LIN {X 0,Y 240.142,Z 967.676,A -85,B 0,C 180,E1 11583.81,E2 11583.81} C_VEL
LIN {X 0,Y 246.627,Z 959.065,A -85,B 0,C 180,E1 11579.011,E2 11579.011} C_VEL
LIN {X 0,Y 253.694,Z 949.494,A -85,B 0,C 180,E1 11574.871,E2 11574.871} C_VEL
LIN {X 0,Y 261.837,Z 937.849,A -85,B 0,C 180,E1 11570.944,E2 11570.944} C_VEL
LIN {X 0,Y 269.961,Z 925.405,A -85,B 0,C 180,E1 11567.617,E2 11567.617} C_VEL
LIN {X 0,Y 278.847,Z 910.719,A -85,B 0,C 180,E1 11564.475,E2 11564.475} C_VEL
LIN {X 0,Y 287.238,Z 895.458,A -85,B 0,C 180,E1 11561.847,E2 11561.847} C_VEL
LIN {X 0,Y 295.186,Z 879.167,A -85,B 0,C 180,E1 11559.593,E2 11559.593} C_VEL
LIN {X 0,Y 302.533,Z 862.052,A -85,B 0,C 180,E1 11557.67,E2 11557.67} C_VEL
LIN {X 0,Y 309.426,Z 843.491,A -85,B 0,C 180,E1 11555.978,E2 11555.978} C_VEL
LIN {X 0,Y 315.478,Z 824.032,A -85,B 0,C 180,E1 11554.564,E2 11554.564} C_VEL
LIN {X 0,Y 320.282,Z 804.619,A -85,B 0,C 180,E1 11553.456,E2 11553.456} C_VEL
LIN {X 0,Y 324.41,Z 782.836,A -85,B 0,C 180,E1 11552.505,E2 11552.505} C_VEL
LIN {X 0,Y 327.137,Z 761.845,A -85,B 0,C 180,E1 11551.838,E2 11551.838} C_VEL
LIN {X 0,Y 332.29,Z 692.537,A -85,B 0,C 180,E1 11550.445,E2 11550.445} C_VEL
LIN {X 0,Y 332.424,Z 684.97,A -85,B 0,C 180,E1 11550.143,E2 11550.143} C_VEL
LIN {X 0,Y 331.311,Z 665.279,A -85,B 0,C 180,E1 11548.776,E2 11548.776} C_VEL
LIN {X 0,Y 331.515,Z 658.771,A -85,B 0,C 180,E1 11548.534,E2 11548.534} C_VEL
LIN {X 0,Y 338.445,Z 571.477,A -85,B 0,C 180,E1 11546.873,E2 11546.873} C_VEL
LIN {X 0,Y 332.872,Z 560.927,A -85,B 0,C 180,E1 11543.609,E2 11543.609} C_VEL
LIN {X 0,Y 328.586,Z 553.31,A -85,B 0,C 180,E1 11540.577,E2 11540.577} C_VEL
LIN {X 0,Y 325.654,Z 548.423,A -85,B 0,C 180,E1 11538.066,E2 11538.066} C_VEL
LIN {X 0,Y 323.732,Z 545.056,A -85,B 0,C 180,E1 11536.047,E2 11536.047} C_VEL
LIN {X 0,Y 321.67,Z 541.505,A -85,B 0,C 180,E1 11533.299,E2 11533.299} C_VEL
LIN {X 0,Y 319.577,Z 537.406,A -85,B 0,C 180,E1 11528.275,E2 11528.275} C_VEL
LIN {X 0,Y 319.566,Z 537.319,A -85,B 0,C 180,E1 11522.87,E2 11522.87} C_VEL
LIN {X 0,Y 320.253,Z 538.098,A -85,B 0,C 180,E1 11520.716,E2 11520.716} C_VEL
LIN {X 0,Y 323.301,Z 542.99,A -85,B 0,C 180,E1 11515.655,E2 11515.655} C_VEL
LIN {X 0,Y 326.289,Z 547.748,A -85,B 0,C 180,E1 11512.517,E2 11512.517} C_VEL
LIN {X 0,Y 329.154,Z 552.402,A -85,B 0,C 180,E1 11510.118,E2 11510.118} C_VEL
LIN {X 0,Y 333.058,Z 558.838,A -85,B 0,C 180,E1 11507.386,E2 11507.386} C_VEL
LIN {X 0,Y 339.072,Z 569.52,A -85,B 0,C 180,E1 11503.864,E2 11503.864} C_VEL
LIN {X 0,Y 341.156,Z 573.867,A -85,B 0,C 180,E1 11502.755,E2 11502.755} C_VEL
LIN {X 0,Y 323.34,Z 778.39,A -85,B 0,C 180,E1 11498.443,E2 11498.443} C_VEL
LIN {X 0,Y 320.486,Z 801.308,A -85,B 0,C 180,E1 11497.861,E2 11497.861} C_VEL
LIN {X 0,Y 316.119,Z 824.113,A -85,B 0,C 180,E1 11497.114,E2 11497.114} C_VEL
LIN {X 0,Y 310.628,Z 846.009,A -85,B 0,C 180,E1 11496.2,E2 11496.2} C_VEL
LIN {X 0,Y 304.335,Z 866.612,A -85,B 0,C 180,E1 11495.063,E2 11495.063} C_VEL
LIN {X 0,Y 296.572,Z 888.375,A -85,B 0,C 180,E1 11493.523,E2 11493.523} C_VEL
LIN {X 0,Y 288.394,Z 908.61,A -85,B 0,C 180,E1 11491.717,E2 11491.717} C_VEL
LIN {X 0,Y 279.584,Z 928.09,A -85,B 0,C 180,E1 11489.528,E2 11489.528} C_VEL
LIN {X 0,Y 270.32,Z 946.899,A -85,B 0,C 180,E1 11486.907,E2 11486.907} C_VEL
LIN {X 0,Y 261.106,Z 964.584,A -85,B 0,C 180,E1 11483.864,E2 11483.864} C_VEL
LIN {X 0,Y 252.022,Z 981.154,A -85,B 0,C 180,E1 11480.324,E2 11480.324} C_VEL
LIN {X 0,Y 243.44,Z 996.518,A -85,B 0,C 180,E1 11476.292,E2 11476.292} C_VEL
LIN {X 0,Y 235.736,Z 1010.633,A -85,B 0,C 180,E1 11471.752,E2 11471.752} C_VEL
LIN {X 0,Y 229.144,Z 1023.261,A -85,B 0,C 180,E1 11466.712,E2 11466.712} C_VEL
LIN {X 0,Y 223.942,Z 1034.477,A -85,B 0,C 180,E1 11461.193,E2 11461.193} C_VEL
LIN {X 0,Y 220.562,Z 1043.412,A -85,B 0,C 180,E1 11455.798,E2 11455.798} C_VEL
LIN {X 0,Y 218.555,Z 1050.849,A -85,B 0,C 180,E1 11450.067,E2 11450.067} C_VEL
LIN {X 0,Y 217.821,Z 1056.561,A -85,B 0,C 180,E1 11444.412,E2 11444.412} C_VEL
LIN {X 0,Y 217.93,Z 1060.05,A -85,B 0,C 180,E1 11439.461,E2 11439.461} C_VEL
LIN {X 0,Y 218.301,Z 1061.983,A -85,B 0,C 180,E1 11435.256,E2 11435.256} C_VEL
LIN {X 0,Y 218.529,Z 1062.818,A -85,B 0,C 180,E1 11431.311,E2 11431.311} C_VEL
LIN {X 0,Y 218.448,Z 1062.621,A -85,B 0,C 180,E1 11427.114,E2 11427.114} C_VEL
LIN {X 0,Y 218.107,Z 1061.202,A -85,B 0,C 180,E1 11422.625,E2 11422.625} C_VEL
LIN {X 0,Y 217.822,Z 1058.052,A -85,B 0,C 180,E1 11417.541,E2 11417.541} C_VEL
LIN {X 0,Y 218.098,Z 1053.522,A -85,B 0,C 180,E1 11412.388,E2 11412.388} C_VEL
LIN {X 0,Y 219.539,Z 1046.762,A -85,B 0,C 180,E1 11406.657,E2 11406.657} C_VEL
LIN {X 0,Y 222.427,Z 1038.271,A -85,B 0,C 180,E1 11400.956,E2 11400.956} C_VEL
LIN {X 0,Y 226.822,Z 1028.031,A -85,B 0,C 180,E1 11395.518,E2 11395.518} C_VEL
LIN {X 0,Y 232.978,Z 1015.73,A -85,B 0,C 180,E1 11390.192,E2 11390.192} C_VEL
LIN {X 0,Y 240.452,Z 1001.951,A -85,B 0,C 180,E1 11385.352,E2 11385.352} C_VEL
LIN {X 0,Y 248.527,Z 987.281,A -85,B 0,C 180,E1 11381.207,E2 11381.207} C_VEL
LIN {X 0,Y 258.12,Z 969.895,A -85,B 0,C 180,E1 11377.222,E2 11377.222} C_VEL
LIN {X 0,Y 267.283,Z 952.769,A -85,B 0,C 180,E1 11374.045,E2 11374.045} C_VEL
LIN {X 0,Y 276.313,Z 934.706,A -85,B 0,C 180,E1 11371.352,E2 11371.352} C_VEL
LIN {X 0,Y 285.607,Z 914.632,A -85,B 0,C 180,E1 11368.93,E2 11368.93} C_VEL
LIN {X 0,Y 294.027,Z 894.724,A -85,B 0,C 180,E1 11367.006,E2 11367.006} C_VEL
LIN {X 0,Y 301.693,Z 874.013,A -85,B 0,C 180,E1 11365.429,E2 11365.429} C_VEL
LIN {X 0,Y 308.866,Z 851.566,A -85,B 0,C 180,E1 11364.091,E2 11364.091} C_VEL
LIN {X 0,Y 314.825,Z 829.345,A -85,B 0,C 180,E1 11363.09,E2 11363.09} C_VEL
LIN {X 0,Y 319.468,Z 806.611,A -85,B 0,C 180,E1 11362.31,E2 11362.31} C_VEL
LIN {X 0,Y 322.699,Z 783.198,A -85,B 0,C 180,E1 11361.682,E2 11361.682} C_VEL
LIN {X 0,Y 339.286,Z 593.485,A -85,B 0,C 180,E1 11357.661,E2 11357.661} C_VEL
LIN {X 0,Y 340.986,Z 573.454,A -85,B 0,C 180,E1 11357.226,E2 11357.226} C_VEL
LIN {X 0,Y 336.419,Z 564.939,A -85,B 0,C 180,E1 11354.764,E2 11354.764} C_VEL
LIN {X 0,Y 331.315,Z 556.08,A -85,B 0,C 180,E1 11351.577,E2 11351.577} C_VEL
LIN {X 0,Y 327.379,Z 549.62,A -85,B 0,C 180,E1 11348.606,E2 11348.606} C_VEL
LIN {X 0,Y 324.756,Z 545.467,A -85,B 0,C 180,E1 11346.186,E2 11346.186} C_VEL
LIN {X 0,Y 322.612,Z 542.052,A -85,B 0,C 180,E1 11343.731,E2 11343.731} C_VEL
LIN {X 0,Y 319.844,Z 537.53,A -85,B 0,C 180,E1 11338.746,E2 11338.746} C_VEL
LIN {X 0,Y 319.024,Z 537,A -85,B 0,C 180,E1 11333.521,E2 11333.521} C_VEL
LIN {X 0,Y 319.531,Z 537.61,A -85,B 0,C 180,E1 11330.817,E2 11330.817} C_VEL
LIN {X 0,Y 322.061,Z 542.358,A -85,B 0,C 180,E1 11325.71,E2 11325.71} C_VEL
LIN {X 0,Y 324.572,Z 546.637,A -85,B 0,C 180,E1 11322.742,E2 11322.742} C_VEL
LIN {X 0,Y 327.505,Z 551.665,A -85,B 0,C 180,E1 11320.056,E2 11320.056} C_VEL
LIN {X 0,Y 331.349,Z 558.399,A -85,B 0,C 180,E1 11317.185,E2 11317.185} C_VEL
LIN {X 0,Y 336.14,Z 567.27,A -85,B 0,C 180,E1 11314.213,E2 11314.213} C_VEL
LIN {X 0,Y 338.286,Z 571.664,A -85,B 0,C 180,E1 11313.017,E2 11313.017} C_VEL
LIN {X 0,Y 323.414,Z 762.056,A -85,B 0,C 180,E1 11309.321,E2 11309.321} C_VEL
LIN {X 0,Y 320.621,Z 783.154,A -85,B 0,C 180,E1 11308.659,E2 11308.659} C_VEL
LIN {X 0,Y 316.72,Z 803.603,A -85,B 0,C 180,E1 11307.786,E2 11307.786} C_VEL
LIN {X 0,Y 311.723,Z 823.559,A -85,B 0,C 180,E1 11306.675,E2 11306.675} C_VEL
LIN {X 0,Y 305.624,Z 842.845,A -85,B 0,C 180,E1 11305.302,E2 11305.302} C_VEL
LIN {X 0,Y 298.738,Z 861.194,A -85,B 0,C 180,E1 11303.671,E2 11303.671} C_VEL
LIN {X 0,Y 291.027,Z 878.909,A -85,B 0,C 180,E1 11301.725,E2 11301.725} C_VEL
LIN {X 0,Y 282.79,Z 895.334,A -85,B 0,C 180,E1 11299.48,E2 11299.48} C_VEL
LIN {X 0,Y 274.659,Z 909.859,A -85,B 0,C 180,E1 11297.031,E2 11297.031} C_VEL
LIN {X 0,Y 265.904,Z 924.109,A -85,B 0,C 180,E1 11294.079,E2 11294.079} C_VEL
LIN {X 0,Y 257.179,Z 937.095,A -85,B 0,C 180,E1 11290.7,E2 11290.7} C_VEL
LIN {X 0,Y 248.83,Z 948.621,A -85,B 0,C 180,E1 11286.904,E2 11286.904} C_VEL
LIN {X 0,Y 240.689,Z 959.299,A -85,B 0,C 180,E1 11282.404,E2 11282.404} C_VEL
LIN {X 0,Y 234.034,Z 967.793,A -85,B 0,C 180,E1 11277.754,E2 11277.754} C_VEL
LIN {X 0,Y 228.325,Z 975.039,A -85,B 0,C 180,E1 11272.482,E2 11272.482} C_VEL
LIN {X 0,Y 224.043,Z 980.52,A -85,B 0,C 180,E1 11266.863,E2 11266.863} C_VEL
LIN {X 0,Y 221.376,Z 984.196,A -85,B 0,C 180,E1 11261.199,E2 11261.199} C_VEL
LIN {X 0,Y 219.974,Z 986.336,A -85,B 0,C 180,E1 11255.471,E2 11255.471} C_VEL
LIN {X 0,Y 219.589,Z 987.052,A -85,B 0,C 180,E1 11250,E2 11250} C_VEL
LIN {X 0,Y 219.961,Z 986.366,A -85,B 0,C 180,E1 11244.522,E2 11244.522} C_VEL
LIN {X 0,Y 221.353,Z 984.268,A -85,B 0,C 180,E1 11238.8,E2 11238.8} C_VEL
LIN {X 0,Y 223.848,Z 980.852,A -85,B 0,C 180,E1 11233.389,E2 11233.389} C_VEL
LIN {X 0,Y 227.962,Z 975.53,A -85,B 0,C 180,E1 11227.839,E2 11227.839} C_VEL
LIN {X 0,Y 233.346,Z 968.696,A -85,B 0,C 180,E1 11222.711,E2 11222.711} C_VEL
LIN {X 0,Y 240.225,Z 959.992,A -85,B 0,C 180,E1 11217.808,E2 11217.808} C_VEL
LIN {X 0,Y 247.681,Z 950.32,A -85,B 0,C 180,E1 11213.6,E2 11213.6} C_VEL
LIN {X 0,Y 256.228,Z 938.614,A -85,B 0,C 180,E1 11209.626,E2 11209.626} C_VEL
LIN {X 0,Y 264.71,Z 926.058,A -85,B 0,C 180,E1 11206.273,E2 11206.273} C_VEL
LIN {X 0,Y 273.954,Z 911.253,A -85,B 0,C 180,E1 11203.118,E2 11203.118} C_VEL
LIN {X 0,Y 282.333,Z 896.481,A -85,B 0,C 180,E1 11200.579,E2 11200.579} C_VEL
LIN {X 0,Y 290.565,Z 880.126,A -85,B 0,C 180,E1 11198.319,E2 11198.319} C_VEL
LIN {X 0,Y 298.139,Z 862.989,A -85,B 0,C 180,E1 11196.401,E2 11196.401} C_VEL
LIN {X 0,Y 305.28,Z 844.29,A -85,B 0,C 180,E1 11194.706,E2 11194.706} C_VEL
LIN {X 0,Y 311.239,Z 825.688,A -85,B 0,C 180,E1 11193.357,E2 11193.357} C_VEL
LIN {X 0,Y 316.405,Z 805.583,A -85,B 0,C 180,E1 11192.209,E2 11192.209} C_VEL
LIN {X 0,Y 320.694,Z 783.638,A -85,B 0,C 180,E1 11191.255,E2 11191.255} C_VEL
LIN {X 0,Y 323.515,Z 762.622,A -85,B 0,C 180,E1 11190.589,E2 11190.589} C_VEL
LIN {X 0,Y 329.217,Z 688.707,A -85,B 0,C 180,E1 11189.11,E2 11189.11} C_VEL
LIN {X 0,Y 331.515,Z 658.771,A -85,B 0,C 180,E1 11188.534,E2 11188.534} C_VEL
LIN {X 0,Y 331.713,Z 651.207,A -85,B 0,C 180,E1 11188.232,E2 11188.232} C_VEL
LIN {X 0,Y 330.89,Z 631.534,A -85,B 0,C 180,E1 11186.847,E2 11186.847} C_VEL
LIN {X 0,Y 331.149,Z 625.029,A -85,B 0,C 180,E1 11186.604,E2 11186.604} C_VEL
LIN {X 0,Y 335.178,Z 576.283,A -85,B 0,C 180,E1 11185.682,E2 11185.682} C_VEL
LIN {X 0,Y 330.368,Z 566.93,A -85,B 0,C 180,E1 11182.652,E2 11182.652} C_VEL
LIN {X 0,Y 326.77,Z 560.37,A -85,B 0,C 180,E1 11179.949,E2 11179.949} C_VEL
LIN {X 0,Y 324.158,Z 555.843,A -85,B 0,C 180,E1 11177.595,E2 11177.595} C_VEL
LIN {X 0,Y 322.398,Z 552.662,A -85,B 0,C 180,E1 11175.654,E2 11175.654} C_VEL
LIN {X 0,Y 320.491,Z 549.259,A -85,B 0,C 180,E1 11172.981,E2 11172.981} C_VEL
LIN {X 0,Y 318.578,Z 545.318,A -85,B 0,C 180,E1 11168.12,E2 11168.12} C_VEL
LIN {X 0,Y 318.631,Z 545.288,A -85,B 0,C 180,E1 11162.698,E2 11162.698} C_VEL
LIN {X 0,Y 319.199,Z 545.972,A -85,B 0,C 180,E1 11160.898,E2 11160.898} C_VEL
LIN {X 0,Y 322.129,Z 550.916,A -85,B 0,C 180,E1 11155.818,E2 11155.818} C_VEL
LIN {X 0,Y 324.879,Z 555.418,A -85,B 0,C 180,E1 11152.84,E2 11152.84} C_VEL
LIN {X 0,Y 327.668,Z 560.099,A -85,B 0,C 180,E1 11150.428,E2 11150.428} C_VEL
LIN {X 0,Y 331.405,Z 566.513,A -85,B 0,C 180,E1 11147.72,E2 11147.72} C_VEL
LIN {X 0,Y 336.99,Z 576.764,A -85,B 0,C 180,E1 11144.336,E2 11144.336} C_VEL
LIN {X 0,Y 337.713,Z 578.605,A -85,B 0,C 180,E1 11143.913,E2 11143.913} C_VEL
LIN {X 0,Y 319.765,Z 778.989,A -85,B 0,C 180,E1 11139.714,E2 11139.714} C_VEL
LIN {X 0,Y 316.751,Z 802.176,A -85,B 0,C 180,E1 11139.125,E2 11139.125} C_VEL
LIN {X 0,Y 312.16,Z 825.001,A -85,B 0,C 180,E1 11138.374,E2 11138.374} C_VEL
LIN {X 0,Y 305.989,Z 848.31,A -85,B 0,C 180,E1 11137.385,E2 11137.385} C_VEL
LIN {X 0,Y 299.382,Z 869.122,A -85,B 0,C 180,E1 11136.219,E2 11136.219} C_VEL
LIN {X 0,Y 291.443,Z 890.215,A -85,B 0,C 180,E1 11134.689,E2 11134.689} C_VEL
LIN {X 0,Y 282.348,Z 911.496,A -85,B 0,C 180,E1 11132.73,E2 11132.73} C_VEL
LIN {X 0,Y 273.35,Z 930.563,A -85,B 0,C 180,E1 11130.524,E2 11130.524} C_VEL
LIN {X 0,Y 263.75,Z 949.037,A -85,B 0,C 180,E1 11127.849,E2 11127.849} C_VEL
LIN {X 0,Y 253.865,Z 966.944,A -85,B 0,C 180,E1 11124.615,E2 11124.615} C_VEL
LIN {X 0,Y 244.481,Z 983.29,A -85,B 0,C 180,E1 11120.964,E2 11120.964} C_VEL
LIN {X 0,Y 235.738,Z 998.112,A -85,B 0,C 180,E1 11116.847,E2 11116.847} C_VEL
LIN {X 0,Y 227.477,Z 1012.397,A -85,B 0,C 180,E1 11111.921,E2 11111.921} C_VEL
LIN {X 0,Y 220.83,Z 1024.643,A -85,B 0,C 180,E1 11106.703,E2 11106.703} C_VEL
LIN {X 0,Y 215.835,Z 1034.911,A -85,B 0,C 180,E1 11101.255,E2 11101.255} C_VEL
LIN {X 0,Y 212.208,Z 1044.211,A -85,B 0,C 180,E1 11095.091,E2 11095.091} C_VEL
LIN {X 0,Y 210.441,Z 1050.98,A -85,B 0,C 180,E1 11089.426,E2 11089.426} C_VEL
LIN {X 0,Y 209.872,Z 1056.146,A -85,B 0,C 180,E1 11083.623,E2 11083.623} C_VEL
LIN {X 0,Y 210.041,Z 1059.081,A -85,B 0,C 180,E1 11079.038,E2 11079.038} C_VEL
LIN {X 0,Y 210.444,Z 1060.875,A -85,B 0,C 180,E1 11074.633,E2 11074.633} C_VEL
LIN {X 0,Y 210.657,Z 1061.576,A -85,B 0,C 180,E1 11070,E2 11070} C_VEL
LIN {X 0,Y 210.447,Z 1060.87,A -85,B 0,C 180,E1 11065.367,E2 11065.367} C_VEL
LIN {X 0,Y 210.042,Z 1059.07,A -85,B 0,C 180,E1 11060.962,E2 11060.962} C_VEL
LIN {X 0,Y 209.875,Z 1056.014,A -85,B 0,C 180,E1 11056.219,E2 11056.219} C_VEL
LIN {X 0,Y 210.5,Z 1050.642,A -85,B 0,C 180,E1 11050.291,E2 11050.291} C_VEL
LIN {X 0,Y 212.286,Z 1043.943,A -85,B 0,C 180,E1 11044.729,E2 11044.729} C_VEL
LIN {X 0,Y 216.045,Z 1034.385,A -85,B 0,C 180,E1 11038.468,E2 11038.468} C_VEL
LIN {X 0,Y 221.119,Z 1024.058,A -85,B 0,C 180,E1 11033.029,E2 11033.029} C_VEL
LIN {X 0,Y 227.849,Z 1011.674,A -85,B 0,C 180,E1 11027.824,E2 11027.824} C_VEL
LIN {X 0,Y 236.185,Z 997.238,A -85,B 0,C 180,E1 11022.914,E2 11022.914} C_VEL
LIN {X 0,Y 245.036,Z 982.255,A -85,B 0,C 180,E1 11018.797,E2 11018.797} C_VEL
LIN {X 0,Y 254.435,Z 965.801,A -85,B 0,C 180,E1 11015.176,E2 11015.176} C_VEL
LIN {X 0,Y 264.307,Z 947.806,A -85,B 0,C 180,E1 11011.978,E2 11011.978} C_VEL
LIN {X 0,Y 273.677,Z 929.711,A -85,B 0,C 180,E1 11009.384,E2 11009.384} C_VEL
LIN {X 0,Y 282.729,Z 910.412,A -85,B 0,C 180,E1 11007.177,E2 11007.177} C_VEL
LIN {X 0,Y 291.431,Z 889.94,A -85,B 0,C 180,E1 11005.306,E2 11005.306} C_VEL
LIN {X 0,Y 298.983,Z 869.874,A -85,B 0,C 180,E1 11003.845,E2 11003.845} C_VEL
LIN {X 0,Y 305.778,Z 848.565,A -85,B 0,C 180,E1 11002.641,E2 11002.641} C_VEL
LIN {X 0,Y 312.057,Z 824.85,A -85,B 0,C 180,E1 11001.634,E2 11001.634} C_VEL
LIN {X 0,Y 316.624,Z 802.081,A -85,B 0,C 180,E1 11000.885,E2 11000.885} C_VEL
LIN {X 0,Y 319.636,Z 778.859,A -85,B 0,C 180,E1 11000.296,E2 11000.296} C_VEL
LIN {X 0,Y 337.501,Z 579.195,A -85,B 0,C 180,E1 10996.11,E2 10996.11} C_VEL
LIN {X 0,Y 337.504,Z 578.002,A -85,B 0,C 180,E1 10996.041,E2 10996.041} C_VEL
LIN {X 0,Y 332.394,Z 568.435,A -85,B 0,C 180,E1 10993.038,E2 10993.038} C_VEL
LIN {X 0,Y 327.928,Z 560.676,A -85,B 0,C 180,E1 10989.919,E2 10989.919} C_VEL
LIN {X 0,Y 325.346,Z 556.368,A -85,B 0,C 180,E1 10987.771,E2 10987.771} C_VEL
LIN {X 0,Y 323.227,Z 552.882,A -85,B 0,C 180,E1 10985.68,E2 10985.68} C_VEL
LIN {X 0,Y 321.331,Z 549.771,A -85,B 0,C 180,E1 10983.389,E2 10983.389} C_VEL
LIN {X 0,Y 318.788,Z 545.43,A -85,B 0,C 180,E1 10978.562,E2 10978.562} C_VEL
LIN {X 0,Y 318.055,Z 544.944,A -85,B 0,C 180,E1 10973.501,E2 10973.501} C_VEL
LIN {X 0,Y 318.512,Z 545.511,A -85,B 0,C 180,E1 10970.969,E2 10970.969} C_VEL
LIN {X 0,Y 320.855,Z 550.07,A -85,B 0,C 180,E1 10966.024,E2 10966.024} C_VEL
LIN {X 0,Y 323.225,Z 554.271,A -85,B 0,C 180,E1 10963.095,E2 10963.095} C_VEL
LIN {X 0,Y 326.081,Z 559.34,A -85,B 0,C 180,E1 10960.381,E2 10960.381} C_VEL
LIN {X 0,Y 329.654,Z 565.803,A -85,B 0,C 180,E1 10957.626,E2 10957.626} C_VEL
LIN {X 0,Y 334.173,Z 574.477,A -85,B 0,C 180,E1 10954.715,E2 10954.715} C_VEL
LIN {X 0,Y 335.017,Z 576.467,A -85,B 0,C 180,E1 10954.203,E2 10954.203} C_VEL
LIN {X 0,Y 319.963,Z 762.597,A -85,B 0,C 180,E1 10950.604,E2 10950.604} C_VEL
LIN {X 0,Y 317.071,Z 783.86,A -85,B 0,C 180,E1 10949.941,E2 10949.941} C_VEL
LIN {X 0,Y 312.847,Z 805.197,A -85,B 0,C 180,E1 10949.032,E2 10949.032} C_VEL
LIN {X 0,Y 307.861,Z 824.509,A -85,B 0,C 180,E1 10947.96,E2 10947.96} C_VEL
LIN {X 0,Y 301.722,Z 843.407,A -85,B 0,C 180,E1 10946.626,E2 10946.626} C_VEL
LIN {X 0,Y 294.37,Z 862.46,A -85,B 0,C 180,E1 10944.944,E2 10944.944} C_VEL
LIN {X 0,Y 286.562,Z 879.874,A -85,B 0,C 180,E1 10943.037,E2 10943.037} C_VEL
LIN {X 0,Y 278.06,Z 896.319,A -85,B 0,C 180,E1 10940.797,E2 10940.797} C_VEL
LIN {X 0,Y 269.358,Z 911.349,A -85,B 0,C 180,E1 10938.255,E2 10938.255} C_VEL
LIN {X 0,Y 260.298,Z 925.555,A -85,B 0,C 180,E1 10935.286,E2 10935.286} C_VEL
LIN {X 0,Y 251.379,Z 938.337,A -85,B 0,C 180,E1 10931.93,E2 10931.93} C_VEL
LIN {X 0,Y 242.745,Z 949.782,A -85,B 0,C 180,E1 10928.119,E2 10928.119} C_VEL
LIN {X 0,Y 234.425,Z 960.224,A -85,B 0,C 180,E1 10923.675,E2 10923.675} C_VEL
LIN {X 0,Y 227.372,Z 968.811,A -85,B 0,C 180,E1 10918.929,E2 10918.929} C_VEL
LIN {X 0,Y 221.416,Z 975.902,A -85,B 0,C 180,E1 10913.697,E2 10913.697} C_VEL
LIN {X 0,Y 216.983,Z 981.232,A -85,B 0,C 180,E1 10908.261,E2 10908.261} C_VEL
LIN {X 0,Y 213.823,Z 985.297,A -85,B 0,C 180,E1 10902.147,E2 10902.147} C_VEL
LIN {X 0,Y 212.264,Z 987.536,A -85,B 0,C 180,E1 10896.491,E2 10896.491} C_VEL
LIN {X 0,Y 211.707,Z 988.358,A -85,B 0,C 180,E1 10890.812,E2 10890.812} C_VEL
LIN {X 0,Y 212.028,Z 987.843,A -85,B 0,C 180,E1 10884.86,E2 10884.86} C_VEL
LIN {X 0,Y 213.416,Z 985.907,A -85,B 0,C 180,E1 10878.925,E2 10878.925} C_VEL
LIN {X 0,Y 216.11,Z 982.432,A -85,B 0,C 180,E1 10873.053,E2 10873.053} C_VEL
LIN {X 0,Y 220.401,Z 977.171,A -85,B 0,C 180,E1 10867.318,E2 10867.318} C_VEL
LIN {X 0,Y 226.02,Z 970.44,A -85,B 0,C 180,E1 10862.036,E2 10862.036} C_VEL
LIN {X 0,Y 233.182,Z 961.85,A -85,B 0,C 180,E1 10857.005,E2 10857.005} C_VEL
LIN {X 0,Y 240.924,Z 952.309,A -85,B 0,C 180,E1 10852.705,E2 10852.705} C_VEL
LIN {X 0,Y 249.762,Z 940.676,A -85,B 0,C 180,E1 10848.659,E2 10848.659} C_VEL
LIN {X 0,Y 258.529,Z 928.292,A -85,B 0,C 180,E1 10845.26,E2 10845.26} C_VEL
LIN {X 0,Y 267.481,Z 914.651,A -85,B 0,C 180,E1 10842.257,E2 10842.257} C_VEL
LIN {X 0,Y 276.393,Z 899.606,A -85,B 0,C 180,E1 10839.598,E2 10839.598} C_VEL
LIN {X 0,Y 284.937,Z 883.381,A -85,B 0,C 180,E1 10837.298,E2 10837.298} C_VEL
LIN {X 0,Y 293.24,Z 865.483,A -85,B 0,C 180,E1 10835.251,E2 10835.251} C_VEL
LIN {X 0,Y 300.578,Z 847.155,A -85,B 0,C 180,E1 10833.562,E2 10833.562} C_VEL
LIN {X 0,Y 307.024,Z 827.711,A -85,B 0,C 180,E1 10832.143,E2 10832.143} C_VEL
LIN {X 0,Y 312.287,Z 808.18,A -85,B 0,C 180,E1 10831.013,E2 10831.013} C_VEL
LIN {X 0,Y 316.625,Z 787.507,A -85,B 0,C 180,E1 10830.087,E2 10830.087} C_VEL
LIN {X 0,Y 319.729,Z 766.245,A -85,B 0,C 180,E1 10829.387,E2 10829.387} C_VEL
LIN {X 0,Y 322.461,Z 733.926,A -85,B 0,C 180,E1 10828.689,E2 10828.689} C_VEL
LIN {X 0,Y 331.149,Z 625.029,A -85,B 0,C 180,E1 10826.604,E2 10826.604} C_VEL
LIN {X 0,Y 331.416,Z 617.467,A -85,B 0,C 180,E1 10826.303,E2 10826.303} C_VEL
LIN {X 0,Y 330.889,Z 597.793,A -85,B 0,C 180,E1 10824.915,E2 10824.915} C_VEL
LIN {X 0,Y 331.198,Z 591.29,A -85,B 0,C 180,E1 10824.673,E2 10824.673} C_VEL
LIN {X 0,Y 332.041,Z 581.053,A -85,B 0,C 180,E1 10824.46,E2 10824.46} C_VEL
LIN {X 0,Y 327.682,Z 572.428,A -85,B 0,C 180,E1 10821.479,E2 10821.479} C_VEL
LIN {X 0,Y 323.761,Z 565.018,A -85,B 0,C 180,E1 10818.175,E2 10818.175} C_VEL
LIN {X 0,Y 321.08,Z 560.265,A -85,B 0,C 180,E1 10815.257,E2 10815.257} C_VEL
LIN {X 0,Y 319.323,Z 557.012,A -85,B 0,C 180,E1 10812.662,E2 10812.662} C_VEL
LIN {X 0,Y 317.577,Z 553.231,A -85,B 0,C 180,E1 10807.963,E2 10807.963} C_VEL
LIN {X 0,Y 317.704,Z 553.262,A -85,B 0,C 180,E1 10802.526,E2 10802.526} C_VEL
LIN {X 0,Y 318.153,Z 553.847,A -85,B 0,C 180,E1 10801.081,E2 10801.081} C_VEL
LIN {X 0,Y 320.907,Z 558.708,A -85,B 0,C 180,E1 10796.07,E2 10796.07} C_VEL
LIN {X 0,Y 323.48,Z 563.088,A -85,B 0,C 180,E1 10793.166,E2 10793.166} C_VEL
LIN {X 0,Y 326.191,Z 567.792,A -85,B 0,C 180,E1 10790.74,E2 10790.74} C_VEL
LIN {X 0,Y 329.83,Z 574.298,A -85,B 0,C 180,E1 10788.016,E2 10788.016} C_VEL
LIN {X 0,Y 334.433,Z 583.129,A -85,B 0,C 180,E1 10785.099,E2 10785.099} C_VEL
LIN {X 0,Y 316.346,Z 779.639,A -85,B 0,C 180,E1 10781.012,E2 10781.012} C_VEL
LIN {X 0,Y 313.22,Z 802.618,A -85,B 0,C 180,E1 10780.429,E2 10780.429} C_VEL
LIN {X 0,Y 308.441,Z 825.524,A -85,B 0,C 180,E1 10779.678,E2 10779.678} C_VEL
LIN {X 0,Y 302.299,Z 847.983,A -85,B 0,C 180,E1 10778.733,E2 10778.733} C_VEL
LIN {X 0,Y 295.336,Z 869.201,A -85,B 0,C 180,E1 10777.555,E2 10777.555} C_VEL
LIN {X 0,Y 287.585,Z 889.224,A -85,B 0,C 180,E1 10776.119,E2 10776.119} C_VEL
LIN {X 0,Y 278.263,Z 910.409,A -85,B 0,C 180,E1 10774.196,E2 10774.196} C_VEL
LIN {X 0,Y 268.934,Z 929.527,A -85,B 0,C 180,E1 10772.006,E2 10772.006} C_VEL
LIN {X 0,Y 259.088,Z 947.794,A -85,B 0,C 180,E1 10769.376,E2 10769.376} C_VEL
LIN {X 0,Y 248.7,Z 965.84,A -85,B 0,C 180,E1 10766.12,E2 10766.12} C_VEL
LIN {X 0,Y 239.204,Z 981.661,A -85,B 0,C 180,E1 10762.579,E2 10762.579} C_VEL
LIN {X 0,Y 229.938,Z 996.555,A -85,B 0,C 180,E1 10758.411,E2 10758.411} C_VEL
LIN {X 0,Y 221.15,Z 1010.865,A -85,B 0,C 180,E1 10753.411,E2 10753.411} C_VEL
LIN {X 0,Y 214.016,Z 1023.136,A -85,B 0,C 180,E1 10748.075,E2 10748.075} C_VEL
LIN {X 0,Y 208.606,Z 1033.416,A -85,B 0,C 180,E1 10742.468,E2 10742.468} C_VEL
LIN {X 0,Y 204.602,Z 1042.743,A -85,B 0,C 180,E1 10736.092,E2 10736.092} C_VEL
LIN {X 0,Y 202.617,Z 1049.532,A -85,B 0,C 180,E1 10730.208,E2 10730.208} C_VEL
LIN {X 0,Y 201.943,Z 1054.611,A -85,B 0,C 180,E1 10724.333,E2 10724.333} C_VEL
LIN {X 0,Y 202.103,Z 1057.687,A -85,B 0,C 180,E1 10719.396,E2 10719.396} C_VEL
LIN {X 0,Y 202.536,Z 1059.501,A -85,B 0,C 180,E1 10714.814,E2 10714.814} C_VEL
LIN {X 0,Y 202.764,Z 1060.193,A -85,B 0,C 180,E1 10710.282,E2 10710.282} C_VEL
LIN {X 0,Y 202.581,Z 1059.672,A -85,B 0,C 180,E1 10705.754,E2 10705.754} C_VEL
LIN {X 0,Y 202.122,Z 1057.825,A -85,B 0,C 180,E1 10700.892,E2 10700.892} C_VEL
LIN {X 0,Y 201.94,Z 1054.805,A -85,B 0,C 180,E1 10695.959,E2 10695.959} C_VEL
LIN {X 0,Y 202.559,Z 1049.825,A -85,B 0,C 180,E1 10690.087,E2 10690.087} C_VEL
LIN {X 0,Y 204.519,Z 1042.949,A -85,B 0,C 180,E1 10684.096,E2 10684.096} C_VEL
LIN {X 0,Y 208.378,Z 1033.853,A -85,B 0,C 180,E1 10677.818,E2 10677.818} C_VEL
LIN {X 0,Y 213.704,Z 1023.627,A -85,B 0,C 180,E1 10672.199,E2 10672.199} C_VEL
LIN {X 0,Y 220.827,Z 1011.333,A -85,B 0,C 180,E1 10666.799,E2 10666.799} C_VEL
LIN {X 0,Y 229.454,Z 997.253,A -85,B 0,C 180,E1 10661.828,E2 10661.828} C_VEL
LIN {X 0,Y 238.652,Z 982.417,A -85,B 0,C 180,E1 10657.642,E2 10657.642} C_VEL
LIN {X 0,Y 248.39,Z 966.219,A -85,B 0,C 180,E1 10653.98,E2 10653.98} C_VEL
LIN {X 0,Y 258.436,Z 948.812,A -85,B 0,C 180,E1 10650.807,E2 10650.807} C_VEL
LIN {X 0,Y 268.223,Z 930.644,A -85,B 0,C 180,E1 10648.162,E2 10648.162} C_VEL
LIN {X 0,Y 277.479,Z 911.808,A -85,B 0,C 180,E1 10645.967,E2 10645.967} C_VEL
LIN {X 0,Y 286.364,Z 891.926,A -85,B 0,C 180,E1 10644.111,E2 10644.111} C_VEL
LIN {X 0,Y 294.139,Z 872.016,A -85,B 0,C 180,E1 10642.645,E2 10642.645} C_VEL
LIN {X 0,Y 301.389,Z 850.49,A -85,B 0,C 180,E1 10641.402,E2 10641.402} C_VEL
LIN {X 0,Y 307.668,Z 828.242,A -85,B 0,C 180,E1 10640.432,E2 10640.432} C_VEL
LIN {X 0,Y 312.541,Z 805.387,A -85,B 0,C 180,E1 10639.669,E2 10639.669} C_VEL
LIN {X 0,Y 315.956,Z 781.829,A -85,B 0,C 180,E1 10639.051,E2 10639.051} C_VEL
LIN {X 0,Y 333.63,Z 590.071,A -85,B 0,C 180,E1 10635.053,E2 10635.053} C_VEL
LIN {X 0,Y 334.211,Z 582.784,A -85,B 0,C 180,E1 10634.864,E2 10634.864} C_VEL
LIN {X 0,Y 328.942,Z 572.781,A -85,B 0,C 180,E1 10631.483,E2 10631.483} C_VEL
LIN {X 0,Y 324.705,Z 565.235,A -85,B 0,C 180,E1 10628.143,E2 10628.143} C_VEL
LIN {X 0,Y 321.96,Z 560.666,A -85,B 0,C 180,E1 10625.435,E2 10625.435} C_VEL
LIN {X 0,Y 320.062,Z 557.488,A -85,B 0,C 180,E1 10623.044,E2 10623.044} C_VEL
LIN {X 0,Y 317.799,Z 553.372,A -85,B 0,C 180,E1 10618.557,E2 10618.557} C_VEL
LIN {X 0,Y 317.086,Z 552.888,A -85,B 0,C 180,E1 10613.481,E2 10613.481} C_VEL
LIN {X 0,Y 317.502,Z 553.412,A -85,B 0,C 180,E1 10611.123,E2 10611.123} C_VEL
LIN {X 0,Y 319.715,Z 557.913,A -85,B 0,C 180,E1 10606.25,E2 10606.25} C_VEL
LIN {X 0,Y 321.937,Z 562.005,A -85,B 0,C 180,E1 10603.397,E2 10603.397} C_VEL
LIN {X 0,Y 324.822,Z 567.273,A -85,B 0,C 180,E1 10600.582,E2 10600.582} C_VEL
LIN {X 0,Y 328.213,Z 573.653,A -85,B 0,C 180,E1 10597.899,E2 10597.899} C_VEL
LIN {X 0,Y 331.918,Z 581.098,A -85,B 0,C 180,E1 10595.415,E2 10595.415} C_VEL
LIN {X 0,Y 316.655,Z 763.362,A -85,B 0,C 180,E1 10591.908,E2 10591.908} C_VEL
LIN {X 0,Y 313.665,Z 784.65,A -85,B 0,C 180,E1 10591.249,E2 10591.249} C_VEL
LIN {X 0,Y 309.431,Z 805.55,A -85,B 0,C 180,E1 10590.369,E2 10590.369} C_VEL
LIN {X 0,Y 304.157,Z 825.454,A -85,B 0,C 180,E1 10589.276,E2 10589.276} C_VEL
LIN {X 0,Y 297.851,Z 844.34,A -85,B 0,C 180,E1 10587.955,E2 10587.955} C_VEL
LIN {X 0,Y 290.29,Z 863.402,A -85,B 0,C 180,E1 10586.286,E2 10586.286} C_VEL
LIN {X 0,Y 282.252,Z 880.838,A -85,B 0,C 180,E1 10584.39,E2 10584.39} C_VEL
LIN {X 0,Y 273.483,Z 897.303,A -85,B 0,C 180,E1 10582.158,E2 10582.158} C_VEL
LIN {X 0,Y 264.185,Z 912.844,A -85,B 0,C 180,E1 10579.528,E2 10579.528} C_VEL
LIN {X 0,Y 254.814,Z 926.999,A -85,B 0,C 180,E1 10576.546,E2 10576.546} C_VEL
LIN {X 0,Y 245.561,Z 939.772,A -85,B 0,C 180,E1 10573.161,E2 10573.161} C_VEL
LIN {X 0,Y 236.637,Z 951.108,A -85,B 0,C 180,E1 10569.331,E2 10569.331} C_VEL
LIN {X 0,Y 227.875,Z 961.618,A -85,B 0,C 180,E1 10564.779,E2 10564.779} C_VEL
LIN {X 0,Y 220.467,Z 970.192,A -85,B 0,C 180,E1 10559.926,E2 10559.926} C_VEL
LIN {X 0,Y 214.177,Z 977.285,A -85,B 0,C 180,E1 10554.55,E2 10554.55} C_VEL
LIN {X 0,Y 209.473,Z 982.607,A -85,B 0,C 180,E1 10548.94,E2 10548.94} C_VEL
LIN {X 0,Y 206.095,Z 986.667,A -85,B 0,C 180,E1 10542.61,E2 10542.61} C_VEL
LIN {X 0,Y 204.422,Z 988.903,A -85,B 0,C 180,E1 10536.741,E2 10536.741} C_VEL
LIN {X 0,Y 203.825,Z 989.723,A -85,B 0,C 180,E1 10530.843,E2 10530.843} C_VEL
LIN {X 0,Y 204.171,Z 989.21,A -85,B 0,C 180,E1 10524.661,E2 10524.661} C_VEL
LIN {X 0,Y 205.661,Z 987.278,A -85,B 0,C 180,E1 10518.502,E2 10518.502} C_VEL
LIN {X 0,Y 208.543,Z 983.803,A -85,B 0,C 180,E1 10512.419,E2 10512.419} C_VEL
LIN {X 0,Y 213.103,Z 978.545,A -85,B 0,C 180,E1 10506.496,E2 10506.496} C_VEL
LIN {X 0,Y 219.048,Z 971.819,A -85,B 0,C 180,E1 10501.063,E2 10501.063} C_VEL
LIN {X 0,Y 226.575,Z 963.239,A -85,B 0,C 180,E1 10495.913,E2 10495.913} C_VEL
LIN {X 0,Y 234.677,Z 953.709,A -85,B 0,C 180,E1 10491.534,E2 10491.534} C_VEL
LIN {X 0,Y 243.884,Z 942.088,A -85,B 0,C 180,E1 10487.432,E2 10487.432} C_VEL
LIN {X 0,Y 252.988,Z 929.736,A -85,B 0,C 180,E1 10484.003,E2 10484.003} C_VEL
LIN {X 0,Y 262.308,Z 916.054,A -85,B 0,C 180,E1 10480.968,E2 10480.968} C_VEL
LIN {X 0,Y 271.452,Z 901.12,A -85,B 0,C 180,E1 10478.32,E2 10478.32} C_VEL
LIN {X 0,Y 280.455,Z 884.589,A -85,B 0,C 180,E1 10475.973,E2 10475.973} C_VEL
LIN {X 0,Y 289.134,Z 866.416,A -85,B 0,C 180,E1 10473.906,E2 10473.906} C_VEL
LIN {X 0,Y 296.68,Z 848.076,A -85,B 0,C 180,E1 10472.23,E2 10472.23} C_VEL
LIN {X 0,Y 303.305,Z 828.634,A -85,B 0,C 180,E1 10470.823,E2 10470.823} C_VEL
LIN {X 0,Y 308.936,Z 808.208,A -85,B 0,C 180,E1 10469.658,E2 10469.658} C_VEL
LIN {X 0,Y 313.406,Z 787.123,A -85,B 0,C 180,E1 10468.737,E2 10468.737} C_VEL
LIN {X 0,Y 316.578,Z 765.801,A -85,B 0,C 180,E1 10468.049,E2 10468.049} C_VEL
LIN {X 0,Y 320.283,Z 722.108,A -85,B 0,C 180,E1 10467.145,E2 10467.145} C_VEL
LIN {X 0,Y 331.198,Z 591.29,A -85,B 0,C 180,E1 10464.673,E2 10464.673} C_VEL
LIN {X 0,Y 331.143,Z 588.442,A -85,B 0,C 180,E1 10464.469,E2 10464.469} C_VEL
LIN {X 0,Y 330.347,Z 585.41,A -85,B 0,C 180,E1 10463.871,E2 10463.871} C_VEL
LIN {X 0,Y 328.792,Z 583.169,A -85,B 0,C 180,E1 10462.889,E2 10462.889} C_VEL
LIN {X 0,Y 326.11,Z 579.993,A -85,B 0,C 180,E1 10461.088,E2 10461.088} C_VEL
LIN {X 0,Y 322.34,Z 572.562,A -85,B 0,C 180,E1 10457.771,E2 10457.771} C_VEL
LIN {X 0,Y 319.846,Z 567.978,A -85,B 0,C 180,E1 10454.946,E2 10454.946} C_VEL
LIN {X 0,Y 318.164,Z 564.762,A -85,B 0,C 180,E1 10452.34,E2 10452.34} C_VEL
LIN {X 0,Y 316.571,Z 561.147,A -85,B 0,C 180,E1 10447.806,E2 10447.806} C_VEL
LIN {X 0,Y 316.728,Z 561.206,A -85,B 0,C 180,E1 10442.534,E2 10442.534} C_VEL
LIN {X 0,Y 317.149,Z 561.901,A -85,B 0,C 180,E1 10441.084,E2 10441.084} C_VEL
LIN {X 0,Y 319.695,Z 566.5,A -85,B 0,C 180,E1 10436.325,E2 10436.325} C_VEL
LIN {X 0,Y 322.186,Z 570.919,A -85,B 0,C 180,E1 10433.407,E2 10433.407} C_VEL
LIN {X 0,Y 324.825,Z 575.665,A -85,B 0,C 180,E1 10430.969,E2 10430.969} C_VEL
LIN {X 0,Y 328.934,Z 583.328,A -85,B 0,C 180,E1 10427.849,E2 10427.849} C_VEL
LIN {X 0,Y 331.247,Z 588.175,A -85,B 0,C 180,E1 10426.297,E2 10426.297} C_VEL
LIN {X 0,Y 313.075,Z 780.483,A -85,B 0,C 180,E1 10422.333,E2 10422.333} C_VEL
LIN {X 0,Y 309.735,Z 803.523,A -85,B 0,C 180,E1 10421.745,E2 10421.745} C_VEL
LIN {X 0,Y 304.892,Z 826.032,A -85,B 0,C 180,E1 10421.014,E2 10421.014} C_VEL
LIN {X 0,Y 298.779,Z 847.657,A -85,B 0,C 180,E1 10420.113,E2 10420.113} C_VEL
LIN {X 0,Y 291.858,Z 868.225,A -85,B 0,C 180,E1 10418.995,E2 10418.995} C_VEL
LIN {X 0,Y 283.91,Z 888.241,A -85,B 0,C 180,E1 10417.588,E2 10417.588} C_VEL
LIN {X 0,Y 274.672,Z 908.705,A -85,B 0,C 180,E1 10415.766,E2 10415.766} C_VEL
LIN {X 0,Y 265.071,Z 927.837,A -85,B 0,C 180,E1 10413.62,E2 10413.62} C_VEL
LIN {X 0,Y 254.871,Z 946.116,A -85,B 0,C 180,E1 10411.025,E2 10411.025} C_VEL
LIN {X 0,Y 244.202,Z 963.97,A -85,B 0,C 180,E1 10407.842,E2 10407.842} C_VEL
LIN {X 0,Y 234.074,Z 980.091,A -85,B 0,C 180,E1 10404.252,E2 10404.252} C_VEL
LIN {X 0,Y 224.327,Z 995.001,A -85,B 0,C 180,E1 10400.053,E2 10400.053} C_VEL
LIN {X 0,Y 214.982,Z 1009.336,A -85,B 0,C 180,E1 10394.987,E2 10394.987} C_VEL
LIN {X 0,Y 207.272,Z 1021.731,A -85,B 0,C 180,E1 10389.484,E2 10389.484} C_VEL
LIN {X 0,Y 201.224,Z 1032.406,A -85,B 0,C 180,E1 10383.473,E2 10383.473} C_VEL
LIN {X 0,Y 197.061,Z 1041.272,A -85,B 0,C 180,E1 10377.171,E2 10377.171} C_VEL
LIN {X 0,Y 194.817,Z 1048.082,A -85,B 0,C 180,E1 10371.055,E2 10371.055} C_VEL
LIN {X 0,Y 194.021,Z 1053.192,A -85,B 0,C 180,E1 10364.932,E2 10364.932} C_VEL
LIN {X 0,Y 194.159,Z 1056.291,A -85,B 0,C 180,E1 10359.784,E2 10359.784} C_VEL
LIN {X 0,Y 194.648,Z 1058.215,A -85,B 0,C 180,E1 10354.714,E2 10354.714} C_VEL
LIN {X 0,Y 194.891,Z 1058.845,A -85,B 0,C 180,E1 10350,E2 10350} C_VEL
LIN {X 0,Y 194.646,Z 1058.188,A -85,B 0,C 180,E1 10345.219,E2 10345.219} C_VEL
LIN {X 0,Y 194.161,Z 1056.279,A -85,B 0,C 180,E1 10340.216,E2 10340.216} C_VEL
LIN {X 0,Y 194.022,Z 1053.174,A -85,B 0,C 180,E1 10335.068,E2 10335.068} C_VEL
LIN {X 0,Y 194.894,Z 1047.739,A -85,B 0,C 180,E1 10328.638,E2 10328.638} C_VEL
LIN {X 0,Y 197.062,Z 1041.24,A -85,B 0,C 180,E1 10322.829,E2 10322.829} C_VEL
LIN {X 0,Y 201.47,Z 1031.875,A -85,B 0,C 180,E1 10316.231,E2 10316.231} C_VEL
LIN {X 0,Y 207.676,Z 1021.029,A -85,B 0,C 180,E1 10310.183,E2 10310.183} C_VEL
LIN {X 0,Y 215.407,Z 1008.607,A -85,B 0,C 180,E1 10304.75,E2 10304.75} C_VEL
LIN {X 0,Y 224.832,Z 994.118,A -85,B 0,C 180,E1 10299.703,E2 10299.703} C_VEL
LIN {X 0,Y 234.638,Z 979.056,A -85,B 0,C 180,E1 10295.52,E2 10295.52} C_VEL
LIN {X 0,Y 244.98,Z 962.58,A -85,B 0,C 180,E1 10291.904,E2 10291.904} C_VEL
LIN {X 0,Y 255.548,Z 944.746,A -85,B 0,C 180,E1 10288.785,E2 10288.785} C_VEL
LIN {X 0,Y 265.735,Z 926.312,A -85,B 0,C 180,E1 10286.216,E2 10286.216} C_VEL
LIN {X 0,Y 275.04,Z 907.681,A -85,B 0,C 180,E1 10284.151,E2 10284.151} C_VEL
LIN {X 0,Y 284.291,Z 886.998,A -85,B 0,C 180,E1 10282.334,E2 10282.334} C_VEL
LIN {X 0,Y 292.251,Z 866.793,A -85,B 0,C 180,E1 10280.932,E2 10280.932} C_VEL
LIN {X 0,Y 299.025,Z 846.405,A -85,B 0,C 180,E1 10279.842,E2 10279.842} C_VEL
LIN {X 0,Y 305.504,Z 822.79,A -85,B 0,C 180,E1 10278.887,E2 10278.887} C_VEL
LIN {X 0,Y 310.19,Z 800.145,A -85,B 0,C 180,E1 10278.172,E2 10278.172} C_VEL
LIN {X 0,Y 313.301,Z 777.065,A -85,B 0,C 180,E1 10277.602,E2 10277.602} C_VEL
LIN {X 0,Y 331.094,Z 587.851,A -85,B 0,C 180,E1 10273.701,E2 10273.701} C_VEL
LIN {X 0,Y 326.753,Z 579.39,A -85,B 0,C 180,E1 10270.713,E2 10270.713} C_VEL
LIN {X 0,Y 323.093,Z 572.603,A -85,B 0,C 180,E1 10267.646,E2 10267.646} C_VEL
LIN {X 0,Y 320.547,Z 568.203,A -85,B 0,C 180,E1 10265.01,E2 10265.01} C_VEL
LIN {X 0,Y 318.923,Z 565.35,A -85,B 0,C 180,E1 10262.875,E2 10262.875} C_VEL
LIN {X 0,Y 316.745,Z 561.272,A -85,B 0,C 180,E1 10258.371,E2 10258.371} C_VEL
LIN {X 0,Y 316.117,Z 560.832,A -85,B 0,C 180,E1 10253.461,E2 10253.461} C_VEL
LIN {X 0,Y 316.537,Z 561.484,A -85,B 0,C 180,E1 10251.096,E2 10251.096} C_VEL
LIN {X 0,Y 318.576,Z 565.755,A -85,B 0,C 180,E1 10246.477,E2 10246.477} C_VEL
LIN {X 0,Y 320.674,Z 569.739,A -85,B 0,C 180,E1 10243.702,E2 10243.702} C_VEL
LIN {X 0,Y 323.38,Z 574.848,A -85,B 0,C 180,E1 10240.961,E2 10240.961} C_VEL
LIN {X 0,Y 326.784,Z 581.492,A -85,B 0,C 180,E1 10238.176,E2 10238.176} C_VEL
LIN {X 0,Y 328.92,Z 586.196,A -85,B 0,C 180,E1 10236.641,E2 10236.641} C_VEL
LIN {X 0,Y 313.524,Z 764.038,A -85,B 0,C 180,E1 10233.241,E2 10233.241} C_VEL
LIN {X 0,Y 310.452,Z 785.291,A -85,B 0,C 180,E1 10232.589,E2 10232.589} C_VEL
LIN {X 0,Y 306.03,Z 806.516,A -85,B 0,C 180,E1 10231.705,E2 10231.705} C_VEL
LIN {X 0,Y 300.617,Z 826.399,A -85,B 0,C 180,E1 10230.625,E2 10230.625} C_VEL
LIN {X 0,Y 293.788,Z 846.245,A -85,B 0,C 180,E1 10229.244,E2 10229.244} C_VEL
LIN {X 0,Y 286.025,Z 865.122,A -85,B 0,C 180,E1 10227.589,E2 10227.589} C_VEL
LIN {X 0,Y 277.761,Z 882.436,A -85,B 0,C 180,E1 10225.704,E2 10225.704} C_VEL
LIN {X 0,Y 268.614,Z 899.085,A -85,B 0,C 180,E1 10223.446,E2 10223.446} C_VEL
LIN {X 0,Y 259.148,Z 914.334,A -85,B 0,C 180,E1 10220.852,E2 10220.852} C_VEL
LIN {X 0,Y 248.869,Z 929.238,A -85,B 0,C 180,E1 10217.667,E2 10217.667} C_VEL
LIN {X 0,Y 239.326,Z 941.902,A -85,B 0,C 180,E1 10214.243,E2 10214.243} C_VEL
LIN {X 0,Y 229.604,Z 953.689,A -85,B 0,C 180,E1 10210.128,E2 10210.128} C_VEL
LIN {X 0,Y 220.991,Z 963.475,A -85,B 0,C 180,E1 10205.708,E2 10205.708} C_VEL
LIN {X 0,Y 213.275,Z 971.935,A -85,B 0,C 180,E1 10200.731,E2 10200.731} C_VEL
LIN {X 0,Y 206.721,Z 978.979,A -85,B 0,C 180,E1 10195.191,E2 10195.191} C_VEL
LIN {X 0,Y 201.606,Z 984.427,A -85,B 0,C 180,E1 10189.107,E2 10189.107} C_VEL
LIN {X 0,Y 198.266,Z 988.173,A -85,B 0,C 180,E1 10182.82,E2 10182.82} C_VEL
LIN {X 0,Y 196.474,Z 990.379,A -85,B 0,C 180,E1 10176.428,E2 10176.428} C_VEL
LIN {X 0,Y 195.941,Z 991.129,A -85,B 0,C 180,E1 10170.292,E2 10170.292} C_VEL
LIN {X 0,Y 196.36,Z 990.52,A -85,B 0,C 180,E1 10164.155,E2 10164.155} C_VEL
LIN {X 0,Y 198.022,Z 988.512,A -85,B 0,C 180,E1 10157.756,E2 10157.756} C_VEL
LIN {X 0,Y 201.185,Z 984.977,A -85,B 0,C 180,E1 10151.454,E2 10151.454} C_VEL
LIN {X 0,Y 206.117,Z 979.654,A -85,B 0,C 180,E1 10145.343,E2 10145.343} C_VEL
LIN {X 0,Y 212.487,Z 972.837,A -85,B 0,C 180,E1 10139.769,E2 10139.769} C_VEL
LIN {X 0,Y 220.472,Z 964.163,A -85,B 0,C 180,E1 10134.515,E2 10134.515} C_VEL
LIN {X 0,Y 229.011,Z 954.54,A -85,B 0,C 180,E1 10130.073,E2 10130.073} C_VEL
LIN {X 0,Y 238.66,Z 942.848,A -85,B 0,C 180,E1 10125.936,E2 10125.936} C_VEL
LIN {X 0,Y 248.153,Z 930.384,A -85,B 0,C 180,E1 10122.494,E2 10122.494} C_VEL
LIN {X 0,Y 257.777,Z 916.67,A -85,B 0,C 180,E1 10119.477,E2 10119.477} C_VEL
LIN {X 0,Y 267.304,Z 901.578,A -85,B 0,C 180,E1 10116.824,E2 10116.824} C_VEL
LIN {X 0,Y 276.261,Z 885.545,A -85,B 0,C 180,E1 10114.575,E2 10114.575} C_VEL
LIN {X 0,Y 285.193,Z 867.349,A -85,B 0,C 180,E1 10112.523,E2 10112.523} C_VEL
LIN {X 0,Y 292.948,Z 848.997,A -85,B 0,C 180,E1 10110.863,E2 10110.863} C_VEL
LIN {X 0,Y 299.751,Z 829.557,A -85,B 0,C 180,E1 10109.471,E2 10109.471} C_VEL
LIN {X 0,Y 305.532,Z 809.159,A -85,B 0,C 180,E1 10108.32,E2 10108.32} C_VEL
LIN {X 0,Y 310.143,Z 788.033,A -85,B 0,C 180,E1 10107.405,E2 10107.405} C_VEL
LIN {X 0,Y 313.43,Z 766.593,A -85,B 0,C 180,E1 10106.719,E2 10106.719} C_VEL
LIN {X 0,Y 317.099,Z 724.828,A -85,B 0,C 180,E1 10105.857,E2 10105.857} C_VEL
LIN {X 0,Y 329.049,Z 585.987,A -85,B 0,C 180,E1 10103.221,E2 10103.221} C_VEL
LIN {X 0,Y 326.11,Z 579.993,A -85,B 0,C 180,E1 10101.088,E2 10101.088} C_VEL
LIN {X 0,Y 324.56,Z 577.933,A -85,B 0,C 180,E1 10099.907,E2 10099.907} C_VEL
LIN {X 0,Y 322.053,Z 577.116,A -85,B 0,C 180,E1 10097.985,E2 10097.985} C_VEL
LIN {X 0,Y 319.338,Z 576.6,A -85,B 0,C 180,E1 10095.506,E2 10095.506} C_VEL
LIN {X 0,Y 318.836,Z 576.035,A -85,B 0,C 180,E1 10094.913,E2 10094.913} C_VEL
LIN {X 0,Y 317.089,Z 572.636,A -85,B 0,C 180,E1 10092.174,E2 10092.174} C_VEL
LIN {X 0,Y 315.567,Z 569.065,A -85,B 0,C 180,E1 10087.648,E2 10087.648} C_VEL
LIN {X 0,Y 315.786,Z 569.187,A -85,B 0,C 180,E1 10082.36,E2 10082.36} C_VEL
LIN {X 0,Y 316.145,Z 569.951,A -85,B 0,C 180,E1 10081.088,E2 10081.088} C_VEL
LIN {X 0,Y 318.49,Z 574.291,A -85,B 0,C 180,E1 10076.581,E2 10076.581} C_VEL
LIN {X 0,Y 320.823,Z 578.588,A -85,B 0,C 180,E1 10073.738,E2 10073.738} C_VEL
LIN {X 0,Y 323.572,Z 583.71,A -85,B 0,C 180,E1 10071.113,E2 10071.113} C_VEL
LIN {X 0,Y 327.289,Z 591.058,A -85,B 0,C 180,E1 10068.19,E2 10068.19} C_VEL
LIN {X 0,Y 328.215,Z 593.242,A -85,B 0,C 180,E1 10067.518,E2 10067.518} C_VEL
LIN {X 0,Y 309.992,Z 781.153,A -85,B 0,C 180,E1 10063.685,E2 10063.685} C_VEL
LIN {X 0,Y 306.273,Z 805.17,A -85,B 0,C 180,E1 10063.068,E2 10063.068} C_VEL
LIN {X 0,Y 301.165,Z 827.894,A -85,B 0,C 180,E1 10062.333,E2 10062.333} C_VEL
LIN {X 0,Y 294.803,Z 849.318,A -85,B 0,C 180,E1 10061.435,E2 10061.435} C_VEL
LIN {X 0,Y 286.919,Z 871.429,A -85,B 0,C 180,E1 10060.205,E2 10060.205} C_VEL
LIN {X 0,Y 278.435,Z 891.883,A -85,B 0,C 180,E1 10058.735,E2 10058.735} C_VEL
LIN {X 0,Y 269.156,Z 911.278,A -85,B 0,C 180,E1 10056.951,E2 10056.951} C_VEL
LIN {X 0,Y 258.446,Z 931.371,A -85,B 0,C 180,E1 10054.602,E2 10054.602} C_VEL
LIN {X 0,Y 248.053,Z 949.191,A -85,B 0,C 180,E1 10051.977,E2 10051.977} C_VEL
LIN {X 0,Y 237.239,Z 966.283,A -85,B 0,C 180,E1 10048.777,E2 10048.777} C_VEL
LIN {X 0,Y 226.203,Z 982.82,A -85,B 0,C 180,E1 10044.859,E2 10044.859} C_VEL
LIN {X 0,Y 216.269,Z 997.305,A -85,B 0,C 180,E1 10040.541,E2 10040.541} C_VEL
LIN {X 0,Y 207.208,Z 1010.436,A -85,B 0,C 180,E1 10035.575,E2 10035.575} C_VEL
LIN {X 0,Y 199.276,Z 1022.428,A -85,B 0,C 180,E1 10029.856,E2 10029.856} C_VEL
LIN {X 0,Y 193.135,Z 1032.799,A -85,B 0,C 180,E1 10023.638,E2 10023.638} C_VEL
LIN {X 0,Y 189.063,Z 1041.002,A -85,B 0,C 180,E1 10017.321,E2 10017.321} C_VEL
LIN {X 0,Y 186.696,Z 1048.052,A -85,B 0,C 180,E1 10010.372,E2 10010.372} C_VEL
LIN {X 0,Y 186.073,Z 1052.402,A -85,B 0,C 180,E1 10004.629,E2 10004.629} C_VEL
LIN {X 0,Y 186.3,Z 1055.498,A -85,B 0,C 180,E1 9998.954,E2 9998.954} C_VEL
LIN {X 0,Y 186.845,Z 1057.108,A -85,B 0,C 180,E1 9993.682,E2 9993.682} C_VEL
LIN {X 0,Y 186.994,Z 1057.408,A -85,B 0,C 180,E1 9989.081,E2 9989.081} C_VEL
LIN {X 0,Y 186.668,Z 1056.646,A -85,B 0,C 180,E1 9984.467,E2 9984.467} C_VEL
LIN {X 0,Y 186.184,Z 1054.657,A -85,B 0,C 180,E1 9979.34,E2 9979.34} C_VEL
LIN {X 0,Y 186.167,Z 1051.115,A -85,B 0,C 180,E1 9973.462,E2 9973.462} C_VEL
LIN {X 0,Y 187.442,Z 1045.332,A -85,B 0,C 180,E1 9966.75,E2 9966.75} C_VEL
LIN {X 0,Y 190.505,Z 1037.882,A -85,B 0,C 180,E1 9960.092,E2 9960.092} C_VEL
LIN {X 0,Y 195.565,Z 1028.452,A -85,B 0,C 180,E1 9953.625,E2 9953.625} C_VEL
LIN {X 0,Y 202.685,Z 1017.126,A -85,B 0,C 180,E1 9947.481,E2 9947.481} C_VEL
LIN {X 0,Y 211.318,Z 1004.422,A -85,B 0,C 180,E1 9942.024,E2 9942.024} C_VEL
LIN {X 0,Y 221.069,Z 990.201,A -85,B 0,C 180,E1 9937.248,E2 9937.248} C_VEL
LIN {X 0,Y 231.598,Z 974.666,A -85,B 0,C 180,E1 9933.118,E2 9933.118} C_VEL
LIN {X 0,Y 242.175,Z 958.518,A -85,B 0,C 180,E1 9929.698,E2 9929.698} C_VEL
LIN {X 0,Y 252.622,Z 941.318,A -85,B 0,C 180,E1 9926.82,E2 9926.82} C_VEL
LIN {X 0,Y 263.685,Z 921.547,A -85,B 0,C 180,E1 9924.197,E2 9924.197} C_VEL
LIN {X 0,Y 273.266,Z 902.726,A -85,B 0,C 180,E1 9922.224,E2 9922.224} C_VEL
LIN {X 0,Y 282.426,Z 882.228,A -85,B 0,C 180,E1 9920.543,E2 9920.543} C_VEL
LIN {X 0,Y 290.617,Z 861.106,A -85,B 0,C 180,E1 9919.193,E2 9919.193} C_VEL
LIN {X 0,Y 297.548,Z 840.24,A -85,B 0,C 180,E1 9918.169,E2 9918.169} C_VEL
LIN {X 0,Y 303.486,Z 817.651,A -85,B 0,C 180,E1 9917.33,E2 9917.33} C_VEL
LIN {X 0,Y 308.024,Z 794.214,A -85,B 0,C 180,E1 9916.645,E2 9916.645} C_VEL
LIN {X 0,Y 311.088,Z 769.502,A -85,B 0,C 180,E1 9916.072,E2 9916.072} C_VEL
LIN {X 0,Y 328.054,Z 592.86,A -85,B 0,C 180,E1 9912.475,E2 9912.475} C_VEL
LIN {X 0,Y 323.799,Z 584.265,A -85,B 0,C 180,E1 9909.239,E2 9909.239} C_VEL
LIN {X 0,Y 320.803,Z 578.738,A -85,B 0,C 180,E1 9906.442,E2 9906.442} C_VEL
LIN {X 0,Y 318.767,Z 575.036,A -85,B 0,C 180,E1 9904.084,E2 9904.084} C_VEL
LIN {X 0,Y 317.553,Z 572.913,A -85,B 0,C 180,E1 9902.345,E2 9902.345} C_VEL
LIN {X 0,Y 315.702,Z 569.171,A -85,B 0,C 180,E1 9898.185,E2 9898.185} C_VEL
LIN {X 0,Y 315.172,Z 568.802,A -85,B 0,C 180,E1 9893.206,E2 9893.206} C_VEL
LIN {X 0,Y 315.526,Z 569.385,A -85,B 0,C 180,E1 9891.25,E2 9891.25} C_VEL
LIN {X 0,Y 317.437,Z 573.595,A -85,B 0,C 180,E1 9886.706,E2 9886.706} C_VEL
LIN {X 0,Y 319.413,Z 577.471,A -85,B 0,C 180,E1 9884.01,E2 9884.01} C_VEL
LIN {X 0,Y 322.24,Z 582.945,A -85,B 0,C 180,E1 9881.079,E2 9881.079} C_VEL
LIN {X 0,Y 325.754,Z 590.226,A -85,B 0,C 180,E1 9878.151,E2 9878.151} C_VEL
LIN {X 0,Y 326.067,Z 591.271,A -85,B 0,C 180,E1 9877.888,E2 9877.888} C_VEL
LIN {X 0,Y 310.563,Z 764.719,A -85,B 0,C 180,E1 9874.599,E2 9874.599} C_VEL
LIN {X 0,Y 307.382,Z 786.109,A -85,B 0,C 180,E1 9873.951,E2 9873.951} C_VEL
LIN {X 0,Y 302.799,Z 807.483,A -85,B 0,C 180,E1 9873.07,E2 9873.07} C_VEL
LIN {X 0,Y 297.248,Z 827.338,A -85,B 0,C 180,E1 9872.005,E2 9872.005} C_VEL
LIN {X 0,Y 290.243,Z 847.175,A -85,B 0,C 180,E1 9870.642,E2 9870.642} C_VEL
LIN {X 0,Y 282.27,Z 866.063,A -85,B 0,C 180,E1 9869.006,E2 9869.006} C_VEL
LIN {X 0,Y 273.772,Z 883.397,A -85,B 0,C 180,E1 9867.14,E2 9867.14} C_VEL
LIN {X 0,Y 264.408,Z 899.964,A -85,B 0,C 180,E1 9864.915,E2 9864.915} C_VEL
LIN {X 0,Y 254.896,Z 914.865,A -85,B 0,C 180,E1 9862.408,E2 9862.408} C_VEL
LIN {X 0,Y 244.853,Z 929.094,A -85,B 0,C 180,E1 9859.424,E2 9859.424} C_VEL
LIN {X 0,Y 234.85,Z 941.92,A -85,B 0,C 180,E1 9856.014,E2 9856.014} C_VEL
LIN {X 0,Y 225.139,Z 953.338,A -85,B 0,C 180,E1 9852.114,E2 9852.114} C_VEL
LIN {X 0,Y 215.5,Z 963.93,A -85,B 0,C 180,E1 9847.431,E2 9847.431} C_VEL
LIN {X 0,Y 207.255,Z 972.588,A -85,B 0,C 180,E1 9842.378,E2 9842.378} C_VEL
LIN {X 0,Y 200.146,Z 979.734,A -85,B 0,C 180,E1 9836.719,E2 9836.719} C_VEL
LIN {X 0,Y 194.763,Z 985.135,A -85,B 0,C 180,E1 9830.746,E2 9830.746} C_VEL
LIN {X 0,Y 190.812,Z 989.273,A -85,B 0,C 180,E1 9823.948,E2 9823.948} C_VEL
LIN {X 0,Y 188.815,Z 991.581,A -85,B 0,C 180,E1 9817.608,E2 9817.608} C_VEL
LIN {X 0,Y 188.067,Z 992.434,A -85,B 0,C 180,E1 9811.219,E2 9811.219} C_VEL
LIN {X 0,Y 188.419,Z 991.998,A -85,B 0,C 180,E1 9804.519,E2 9804.519} C_VEL
LIN {X 0,Y 189.975,Z 990.29,A -85,B 0,C 180,E1 9798.155,E2 9798.155} C_VEL
LIN {X 0,Y 193.112,Z 986.899,A -85,B 0,C 180,E1 9791.589,E2 9791.589} C_VEL
LIN {X 0,Y 198.11,Z 981.829,A -85,B 0,C 180,E1 9785.235,E2 9785.235} C_VEL
LIN {X 0,Y 205.05,Z 974.85,A -85,B 0,C 180,E1 9779.117,E2 9779.117} C_VEL
LIN {X 0,Y 213.206,Z 966.49,A -85,B 0,C 180,E1 9773.779,E2 9773.779} C_VEL
LIN {X 0,Y 222.501,Z 956.497,A -85,B 0,C 180,E1 9768.998,E2 9768.998} C_VEL
LIN {X 0,Y 232.49,Z 944.911,A -85,B 0,C 180,E1 9764.796,E2 9764.796} C_VEL
LIN {X 0,Y 242.896,Z 931.827,A -85,B 0,C 180,E1 9761.122,E2 9761.122} C_VEL
LIN {X 0,Y 253.484,Z 917.199,A -85,B 0,C 180,E1 9757.917,E2 9757.917} C_VEL
LIN {X 0,Y 263.343,Z 902.034,A -85,B 0,C 180,E1 9755.282,E2 9755.282} C_VEL
LIN {X 0,Y 272.645,Z 885.749,A -85,B 0,C 180,E1 9753.04,E2 9753.04} C_VEL
LIN {X 0,Y 281.778,Z 867.5,A -85,B 0,C 180,E1 9751.025,E2 9751.025} C_VEL
LIN {X 0,Y 289.749,Z 848.945,A -85,B 0,C 180,E1 9749.387,E2 9749.387} C_VEL
LIN {X 0,Y 296.741,Z 829.377,A -85,B 0,C 180,E1 9748.017,E2 9748.017} C_VEL
LIN {X 0,Y 302.363,Z 809.84,A -85,B 0,C 180,E1 9746.939,E2 9746.939} C_VEL
LIN {X 0,Y 307.093,Z 788.684,A -85,B 0,C 180,E1 9746.036,E2 9746.036} C_VEL
LIN {X 0,Y 310.482,Z 767.177,A -85,B 0,C 180,E1 9745.357,E2 9745.357} C_VEL
LIN {X 0,Y 314.389,Z 724.052,A -85,B 0,C 180,E1 9744.477,E2 9744.477} C_VEL
LIN {X 0,Y 326.263,Z 591.09,A -85,B 0,C 180,E1 9742.003,E2 9742.003} C_VEL
LIN {X 0,Y 322.539,Z 583.363,A -85,B 0,C 180,E1 9738.949,E2 9738.949} C_VEL
LIN {X 0,Y 319.672,Z 577.781,A -85,B 0,C 180,E1 9735.977,E2 9735.977} C_VEL
LIN {X 0,Y 318.836,Z 576.035,A -85,B 0,C 180,E1 9734.913,E2 9734.913} C_VEL
LIN {X 0,Y 317.725,Z 575.445,A -85,B 0,C 180,E1 9733.533,E2 9733.533} C_VEL
LIN {X 0,Y 315.051,Z 577.948,A -85,B 0,C 180,E1 9729.523,E2 9729.523} C_VEL
LIN {X 0,Y 314.748,Z 577.561,A -85,B 0,C 180,E1 9728.511,E2 9728.511} C_VEL
LIN {X 0,Y 314.479,Z 576.923,A -85,B 0,C 180,E1 9726.94,E2 9726.94} C_VEL
LIN {X 0,Y 314.899,Z 577.213,A -85,B 0,C 180,E1 9722.002,E2 9722.002} C_VEL
LIN {X 0,Y 317.284,Z 582.081,A -85,B 0,C 180,E1 9716.839,E2 9716.839} C_VEL
LIN {X 0,Y 319.454,Z 586.255,A -85,B 0,C 180,E1 9714.072,E2 9714.072} C_VEL
LIN {X 0,Y 322.365,Z 591.836,A -85,B 0,C 180,E1 9711.214,E2 9711.214} C_VEL
LIN {X 0,Y 325.34,Z 598.219,A -85,B 0,C 180,E1 9708.762,E2 9708.762} C_VEL
LIN {X 0,Y 307.15,Z 781.329,A -85,B 0,C 180,E1 9705.075,E2 9705.075} C_VEL
LIN {X 0,Y 303.263,Z 805.417,A -85,B 0,C 180,E1 9704.462,E2 9704.462} C_VEL
LIN {X 0,Y 298.115,Z 827.652,A -85,B 0,C 180,E1 9703.755,E2 9703.755} C_VEL
LIN {X 0,Y 291.56,Z 849.231,A -85,B 0,C 180,E1 9702.87,E2 9702.87} C_VEL
LIN {X 0,Y 283.636,Z 870.844,A -85,B 0,C 180,E1 9701.693,E2 9701.693} C_VEL
LIN {X 0,Y 275.094,Z 890.92,A -85,B 0,C 180,E1 9700.283,E2 9700.283} C_VEL
LIN {X 0,Y 265.973,Z 909.511,A -85,B 0,C 180,E1 9698.615,E2 9698.615} C_VEL
LIN {X 0,Y 255.013,Z 929.558,A -85,B 0,C 180,E1 9696.336,E2 9696.336} C_VEL
LIN {X 0,Y 244.174,Z 947.576,A -85,B 0,C 180,E1 9693.738,E2 9693.738} C_VEL
LIN {X 0,Y 232.65,Z 965.088,A -85,B 0,C 180,E1 9690.492,E2 9690.492} C_VEL
LIN {X 0,Y 221.363,Z 981.254,A -85,B 0,C 180,E1 9686.68,E2 9686.68} C_VEL
LIN {X 0,Y 210.741,Z 996,A -85,B 0,C 180,E1 9682.264,E2 9682.264} C_VEL
LIN {X 0,Y 200.818,Z 1009.562,A -85,B 0,C 180,E1 9677.047,E2 9677.047} C_VEL
LIN {X 0,Y 192.504,Z 1021.316,A -85,B 0,C 180,E1 9671.272,E2 9671.272} C_VEL
LIN {X 0,Y 185.833,Z 1031.744,A -85,B 0,C 180,E1 9664.773,E2 9664.773} C_VEL
LIN {X 0,Y 181.385,Z 1040.009,A -85,B 0,C 180,E1 9658.12,E2 9658.12} C_VEL
LIN {X 0,Y 178.836,Z 1046.876,A -85,B 0,C 180,E1 9650.966,E2 9650.966} C_VEL
LIN {X 0,Y 178.142,Z 1051.192,A -85,B 0,C 180,E1 9644.962,E2 9644.962} C_VEL
LIN {X 0,Y 178.407,Z 1054.378,A -85,B 0,C 180,E1 9638.703,E2 9638.703} C_VEL
LIN {X 0,Y 178.969,Z 1055.776,A -85,B 0,C 180,E1 9633.523,E2 9633.523} C_VEL
LIN {X 0,Y 179.11,Z 1056.042,A -85,B 0,C 180,E1 9629.04,E2 9629.04} C_VEL
LIN {X 0,Y 178.774,Z 1055.36,A -85,B 0,C 180,E1 9624.544,E2 9624.544} C_VEL
LIN {X 0,Y 178.264,Z 1053.479,A -85,B 0,C 180,E1 9619.333,E2 9619.333} C_VEL
LIN {X 0,Y 178.213,Z 1050.265,A -85,B 0,C 180,E1 9613.611,E2 9613.611} C_VEL
LIN {X 0,Y 179.447,Z 1044.831,A -85,B 0,C 180,E1 9606.696,E2 9606.696} C_VEL
LIN {X 0,Y 182.447,Z 1037.816,A -85,B 0,C 180,E1 9599.981,E2 9599.981} C_VEL
LIN {X 0,Y 187.824,Z 1028.4,A -85,B 0,C 180,E1 9593.019,E2 9593.019} C_VEL
LIN {X 0,Y 194.815,Z 1017.992,A -85,B 0,C 180,E1 9586.952,E2 9586.952} C_VEL
LIN {X 0,Y 203.668,Z 1005.551,A -85,B 0,C 180,E1 9581.312,E2 9581.312} C_VEL
LIN {X 0,Y 213.683,Z 991.792,A -85,B 0,C 180,E1 9576.407,E2 9576.407} C_VEL
LIN {X 0,Y 224.471,Z 976.808,A -85,B 0,C 180,E1 9572.186,E2 9572.186} C_VEL
LIN {X 0,Y 235.71,Z 960.387,A -85,B 0,C 180,E1 9568.588,E2 9568.588} C_VEL
LIN {X 0,Y 247.08,Z 942.626,A -85,B 0,C 180,E1 9565.522,E2 9565.522} C_VEL
LIN {X 0,Y 257.683,Z 924.719,A -85,B 0,C 180,E1 9563.072,E2 9563.072} C_VEL
LIN {X 0,Y 267.797,Z 905.66,A -85,B 0,C 180,E1 9561.026,E2 9561.026} C_VEL
LIN {X 0,Y 277.542,Z 885.011,A -85,B 0,C 180,E1 9559.287,E2 9559.287} C_VEL
LIN {X 0,Y 285.887,Z 864.81,A -85,B 0,C 180,E1 9557.955,E2 9557.955} C_VEL
LIN {X 0,Y 293.133,Z 843.911,A -85,B 0,C 180,E1 9556.907,E2 9556.907} C_VEL
LIN {X 0,Y 299.694,Z 820.702,A -85,B 0,C 180,E1 9556.024,E2 9556.024} C_VEL
LIN {X 0,Y 304.505,Z 798.081,A -85,B 0,C 180,E1 9555.346,E2 9555.346} C_VEL
LIN {X 0,Y 307.701,Z 775.17,A -85,B 0,C 180,E1 9554.801,E2 9554.801} C_VEL
LIN {X 0,Y 325.184,Z 597.949,A -85,B 0,C 180,E1 9551.236,E2 9551.236} C_VEL
LIN {X 0,Y 321.639,Z 590.704,A -85,B 0,C 180,E1 9548.311,E2 9548.311} C_VEL
LIN {X 0,Y 318.817,Z 585.106,A -85,B 0,C 180,E1 9545.398,E2 9545.398} C_VEL
LIN {X 0,Y 316.552,Z 580.929,A -85,B 0,C 180,E1 9542.353,E2 9542.353} C_VEL
LIN {X 0,Y 314.67,Z 577.072,A -85,B 0,C 180,E1 9537.996,E2 9537.996} C_VEL
LIN {X 0,Y 314.219,Z 576.759,A -85,B 0,C 180,E1 9533.054,E2 9533.054} C_VEL
LIN {X 0,Y 314.518,Z 577.316,A -85,B 0,C 180,E1 9531.373,E2 9531.373} C_VEL
LIN {X 0,Y 316.26,Z 581.305,A -85,B 0,C 180,E1 9527.028,E2 9527.028} C_VEL
LIN {X 0,Y 318.081,Z 585.04,A -85,B 0,C 180,E1 9524.409,E2 9524.409} C_VEL
LIN {X 0,Y 320.809,Z 590.517,A -85,B 0,C 180,E1 9521.463,E2 9521.463} C_VEL
LIN {X 0,Y 323.393,Z 596.272,A -85,B 0,C 180,E1 9519.159,E2 9519.159} C_VEL
LIN {X 0,Y 307.768,Z 765.506,A -85,B 0,C 180,E1 9515.981,E2 9515.981} C_VEL
LIN {X 0,Y 304.504,Z 786.825,A -85,B 0,C 180,E1 9515.343,E2 9515.343} C_VEL
LIN {X 0,Y 299.937,Z 807.725,A -85,B 0,C 180,E1 9514.498,E2 9514.498} C_VEL
LIN {X 0,Y 294.43,Z 827.033,A -85,B 0,C 180,E1 9513.487,E2 9513.487} C_VEL
LIN {X 0,Y 287.662,Z 846.063,A -85,B 0,C 180,E1 9512.224,E2 9512.224} C_VEL
LIN {X 0,Y 279.431,Z 865.439,A -85,B 0,C 180,E1 9510.61,E2 9510.61} C_VEL
LIN {X 0,Y 270.687,Z 883.057,A -85,B 0,C 180,E1 9508.773,E2 9508.773} C_VEL
LIN {X 0,Y 261.09,Z 899.658,A -85,B 0,C 180,E1 9506.6,E2 9506.6} C_VEL
LIN {X 0,Y 250.84,Z 915.4,A -85,B 0,C 180,E1 9504.015,E2 9504.015} C_VEL
LIN {X 0,Y 240.439,Z 929.742,A -85,B 0,C 180,E1 9501.045,E2 9501.045} C_VEL
LIN {X 0,Y 230.01,Z 942.647,A -85,B 0,C 180,E1 9497.639,E2 9497.639} C_VEL
LIN {X 0,Y 219.652,Z 954.395,A -85,B 0,C 180,E1 9493.632,E2 9493.632} C_VEL
LIN {X 0,Y 209.737,Z 964.85,A -85,B 0,C 180,E1 9488.997,E2 9488.997} C_VEL
LIN {X 0,Y 200.885,Z 973.714,A -85,B 0,C 180,E1 9483.776,E2 9483.776} C_VEL
LIN {X 0,Y 193.095,Z 981.116,A -85,B 0,C 180,E1 9477.777,E2 9477.777} C_VEL
LIN {X 0,Y 187.373,Z 986.51,A -85,B 0,C 180,E1 9471.605,E2 9471.605} C_VEL
LIN {X 0,Y 183.142,Z 990.643,A -85,B 0,C 180,E1 9464.545,E2 9464.545} C_VEL
LIN {X 0,Y 180.992,Z 992.948,A -85,B 0,C 180,E1 9457.938,E2 9457.938} C_VEL
LIN {X 0,Y 180.185,Z 993.8,A -85,B 0,C 180,E1 9451.272,E2 9451.272} C_VEL
LIN {X 0,Y 180.567,Z 993.365,A -85,B 0,C 180,E1 9444.28,E2 9444.28} C_VEL
LIN {X 0,Y 182.291,Z 991.603,A -85,B 0,C 180,E1 9437.512,E2 9437.512} C_VEL
LIN {X 0,Y 185.812,Z 988.092,A -85,B 0,C 180,E1 9430.511,E2 9430.511} C_VEL
LIN {X 0,Y 190.934,Z 983.202,A -85,B 0,C 180,E1 9424.237,E2 9424.237} C_VEL
LIN {X 0,Y 198.189,Z 976.323,A -85,B 0,C 180,E1 9418.013,E2 9418.013} C_VEL
LIN {X 0,Y 206.42,Z 968.348,A -85,B 0,C 180,E1 9412.737,E2 9412.737} C_VEL
LIN {X 0,Y 216.068,Z 958.416,A -85,B 0,C 180,E1 9407.856,E2 9407.856} C_VEL
LIN {X 0,Y 226.416,Z 946.972,A -85,B 0,C 180,E1 9403.595,E2 9403.595} C_VEL
LIN {X 0,Y 237.452,Z 933.689,A -85,B 0,C 180,E1 9399.796,E2 9399.796} C_VEL
LIN {X 0,Y 248.069,Z 919.641,A -85,B 0,C 180,E1 9396.67,E2 9396.67} C_VEL
LIN {X 0,Y 258.19,Z 904.6,A -85,B 0,C 180,E1 9394.031,E2 9394.031} C_VEL
LIN {X 0,Y 268.031,Z 888.088,A -85,B 0,C 180,E1 9391.73,E2 9391.73} C_VEL
LIN {X 0,Y 277.017,Z 870.939,A -85,B 0,C 180,E1 9389.812,E2 9389.812} C_VEL
LIN {X 0,Y 285.252,Z 852.621,A -85,B 0,C 180,E1 9388.169,E2 9388.169} C_VEL
LIN {X 0,Y 292.4,Z 833.582,A -85,B 0,C 180,E1 9386.812,E2 9386.812} C_VEL
LIN {X 0,Y 298.857,Z 812.484,A -85,B 0,C 180,E1 9385.624,E2 9385.624} C_VEL
LIN {X 0,Y 303.783,Z 791.746,A -85,B 0,C 180,E1 9384.726,E2 9384.726} C_VEL
LIN {X 0,Y 307.361,Z 770.158,A -85,B 0,C 180,E1 9384.035,E2 9384.035} C_VEL
LIN {X 0,Y 310.369,Z 740.148,A -85,B 0,C 180,E1 9383.388,E2 9383.388} C_VEL
LIN {X 0,Y 323.56,Z 596.216,A -85,B 0,C 180,E1 9380.731,E2 9380.731} C_VEL
LIN {X 0,Y 320.413,Z 589.612,A -85,B 0,C 180,E1 9377.901,E2 9377.901} C_VEL
LIN {X 0,Y 317.672,Z 583.844,A -85,B 0,C 180,E1 9374.678,E2 9374.678} C_VEL
LIN {X 0,Y 315.948,Z 580.402,A -85,B 0,C 180,E1 9371.871,E2 9371.871} C_VEL
LIN {X 0,Y 314.748,Z 577.561,A -85,B 0,C 180,E1 9368.511,E2 9368.511} C_VEL
LIN {X 0,Y 314.467,Z 577.521,A -85,B 0,C 180,E1 9367.309,E2 9367.309} C_VEL
LIN {X 0,Y 314.015,Z 579.84,A -85,B 0,C 180,E1 9365.636,E2 9365.636} C_VEL
LIN {X 0,Y 313.718,Z 584.426,A -85,B 0,C 180,E1 9363.072,E2 9363.072} C_VEL
LIN {X 0,Y 313.88,Z 585.125,A -85,B 0,C 180,E1 9362.152,E2 9362.152} C_VEL
LIN {X 0,Y 316.085,Z 589.87,A -85,B 0,C 180,E1 9357.099,E2 9357.099} C_VEL
LIN {X 0,Y 318.095,Z 593.92,A -85,B 0,C 180,E1 9354.409,E2 9354.409} C_VEL
LIN {X 0,Y 320.856,Z 599.48,A -85,B 0,C 180,E1 9351.579,E2 9351.579} C_VEL
LIN {X 0,Y 322.609,Z 603.49,A -85,B 0,C 180,E1 9350.023,E2 9350.023} C_VEL
LIN {X 0,Y 304.377,Z 782.447,A -85,B 0,C 180,E1 9346.47,E2 9346.47} C_VEL
LIN {X 0,Y 300.468,Z 805.523,A -85,B 0,C 180,E1 9345.887,E2 9345.887} C_VEL
LIN {X 0,Y 295.119,Z 827.865,A -85,B 0,C 180,E1 9345.188,E2 9345.188} C_VEL
LIN {X 0,Y 288.654,Z 848.689,A -85,B 0,C 180,E1 9344.357,E2 9344.357} C_VEL
LIN {X 0,Y 280.632,Z 870.06,A -85,B 0,C 180,E1 9343.227,E2 9343.227} C_VEL
LIN {X 0,Y 271.969,Z 889.941,A -85,B 0,C 180,E1 9341.869,E2 9341.869} C_VEL
LIN {X 0,Y 262.459,Z 908.818,A -85,B 0,C 180,E1 9340.216,E2 9340.216} C_VEL
LIN {X 0,Y 251.268,Z 928.661,A -85,B 0,C 180,E1 9337.999,E2 9337.999} C_VEL
LIN {X 0,Y 240.163,Z 946.516,A -85,B 0,C 180,E1 9335.461,E2 9335.461} C_VEL
LIN {X 0,Y 228.687,Z 963.318,A -85,B 0,C 180,E1 9332.391,E2 9332.391} C_VEL
LIN {X 0,Y 216.763,Z 979.691,A -85,B 0,C 180,E1 9328.578,E2 9328.578} C_VEL
LIN {X 0,Y 205.777,Z 994.242,A -85,B 0,C 180,E1 9324.238,E2 9324.238} C_VEL
LIN {X 0,Y 195.387,Z 1007.606,A -85,B 0,C 180,E1 9319.08,E2 9319.08} C_VEL
LIN {X 0,Y 186.15,Z 1019.81,A -85,B 0,C 180,E1 9313.012,E2 9313.012} C_VEL
LIN {X 0,Y 178.895,Z 1030.26,A -85,B 0,C 180,E1 9306.331,E2 9306.331} C_VEL
LIN {X 0,Y 173.889,Z 1038.728,A -85,B 0,C 180,E1 9299.259,E2 9299.259} C_VEL
LIN {X 0,Y 170.992,Z 1045.703,A -85,B 0,C 180,E1 9291.609,E2 9291.609} C_VEL
LIN {X 0,Y 170.215,Z 1049.981,A -85,B 0,C 180,E1 9285.327,E2 9285.327} C_VEL
LIN {X 0,Y 170.492,Z 1053.089,A -85,B 0,C 180,E1 9278.771,E2 9278.771} C_VEL
LIN {X 0,Y 171.093,Z 1054.444,A -85,B 0,C 180,E1 9273.35,E2 9273.35} C_VEL
LIN {X 0,Y 171.225,Z 1054.676,A -85,B 0,C 180,E1 9268.996,E2 9268.996} C_VEL
LIN {X 0,Y 170.836,Z 1053.964,A -85,B 0,C 180,E1 9264.237,E2 9264.237} C_VEL
LIN {X 0,Y 170.307,Z 1051.991,A -85,B 0,C 180,E1 9258.644,E2 9258.644} C_VEL
LIN {X 0,Y 170.369,Z 1048.469,A -85,B 0,C 180,E1 9252.231,E2 9252.231} C_VEL
LIN {X 0,Y 172.042,Z 1042.738,A -85,B 0,C 180,E1 9244.896,E2 9244.896} C_VEL
LIN {X 0,Y 175.764,Z 1035.323,A -85,B 0,C 180,E1 9237.674,E2 9237.674} C_VEL
LIN {X 0,Y 181.731,Z 1025.938,A -85,B 0,C 180,E1 9230.749,E2 9230.749} C_VEL
LIN {X 0,Y 190.37,Z 1014.087,A -85,B 0,C 180,E1 9223.982,E2 9223.982} C_VEL
LIN {X 0,Y 200.2,Z 1001.331,A -85,B 0,C 180,E1 9218.361,E2 9218.361} C_VEL
LIN {X 0,Y 211.118,Z 987.103,A -85,B 0,C 180,E1 9213.535,E2 9213.535} C_VEL
LIN {X 0,Y 222.705,Z 971.501,A -85,B 0,C 180,E1 9209.426,E2 9209.426} C_VEL
LIN {X 0,Y 234.013,Z 955.503,A -85,B 0,C 180,E1 9206.108,E2 9206.108} C_VEL
LIN {X 0,Y 245.438,Z 937.989,A -85,B 0,C 180,E1 9203.275,E2 9203.275} C_VEL
LIN {X 0,Y 256.783,Z 918.858,A -85,B 0,C 180,E1 9200.85,E2 9200.85} C_VEL
LIN {X 0,Y 267.366,Z 899.014,A -85,B 0,C 180,E1 9198.889,E2 9198.889} C_VEL
LIN {X 0,Y 277.053,Z 878.281,A -85,B 0,C 180,E1 9197.303,E2 9197.303} C_VEL
LIN {X 0,Y 285.457,Z 857.147,A -85,B 0,C 180,E1 9196.063,E2 9196.063} C_VEL
LIN {X 0,Y 293.031,Z 834.417,A -85,B 0,C 180,E1 9195.063,E2 9195.063} C_VEL
LIN {X 0,Y 298.989,Z 811.851,A -85,B 0,C 180,E1 9194.304,E2 9194.304} C_VEL
LIN {X 0,Y 303.283,Z 788.856,A -85,B 0,C 180,E1 9193.691,E2 9193.691} C_VEL
LIN {X 0,Y 307.009,Z 756.365,A -85,B 0,C 180,E1 9192.998,E2 9192.998} C_VEL
LIN {X 0,Y 322.418,Z 603.108,A -85,B 0,C 180,E1 9189.955,E2 9189.955} C_VEL
LIN {X 0,Y 319.228,Z 596.349,A -85,B 0,C 180,E1 9187.016,E2 9187.016} C_VEL
LIN {X 0,Y 316.704,Z 591.313,A -85,B 0,C 180,E1 9184.073,E2 9184.073} C_VEL
LIN {X 0,Y 315.209,Z 588.487,A -85,B 0,C 180,E1 9181.817,E2 9181.817} C_VEL
LIN {X 0,Y 313.64,Z 584.973,A -85,B 0,C 180,E1 9177.807,E2 9177.807} C_VEL
LIN {X 0,Y 313.275,Z 584.722,A -85,B 0,C 180,E1 9172.849,E2 9172.849} C_VEL
LIN {X 0,Y 313.532,Z 585.353,A -85,B 0,C 180,E1 9171.379,E2 9171.379} C_VEL
LIN {X 0,Y 315.142,Z 589.144,A -85,B 0,C 180,E1 9167.261,E2 9167.261} C_VEL
LIN {X 0,Y 316.831,Z 592.769,A -85,B 0,C 180,E1 9164.721,E2 9164.721} C_VEL
LIN {X 0,Y 319.421,Z 598.209,A -85,B 0,C 180,E1 9161.805,E2 9161.805} C_VEL
LIN {X 0,Y 320.827,Z 601.639,A -85,B 0,C 180,E1 9160.442,E2 9160.442} C_VEL
LIN {X 0,Y 305.19,Z 765.994,A -85,B 0,C 180,E1 9157.395,E2 9157.395} C_VEL
LIN {X 0,Y 301.826,Z 787.452,A -85,B 0,C 180,E1 9156.763,E2 9156.763} C_VEL
LIN {X 0,Y 297.067,Z 808.682,A -85,B 0,C 180,E1 9155.92,E2 9155.92} C_VEL
LIN {X 0,Y 291.429,Z 827.971,A -85,B 0,C 180,E1 9154.926,E2 9154.926} C_VEL
LIN {X 0,Y 284.457,Z 847.087,A -85,B 0,C 180,E1 9153.679,E2 9153.679} C_VEL
LIN {X 0,Y 276.057,Z 866.375,A -85,B 0,C 180,E1 9152.099,E2 9152.099} C_VEL
LIN {X 0,Y 267.079,Z 884.008,A -85,B 0,C 180,E1 9150.29,E2 9150.29} C_VEL
LIN {X 0,Y 257.212,Z 900.631,A -85,B 0,C 180,E1 9148.145,E2 9148.145} C_VEL
LIN {X 0,Y 246.299,Z 916.884,A -85,B 0,C 180,E1 9145.497,E2 9145.497} C_VEL
LIN {X 0,Y 235.563,Z 931.183,A -85,B 0,C 180,E1 9142.536,E2 9142.536} C_VEL
LIN {X 0,Y 224.173,Z 944.785,A -85,B 0,C 180,E1 9138.919,E2 9138.919} C_VEL
LIN {X 0,Y 213.672,Z 956.148,A -85,B 0,C 180,E1 9134.959,E2 9134.959} C_VEL
LIN {X 0,Y 203.147,Z 966.707,A -85,B 0,C 180,E1 9130.148,E2 9130.148} C_VEL
LIN {X 0,Y 194.05,Z 975.347,A -85,B 0,C 180,E1 9124.886,E2 9124.886} C_VEL
LIN {X 0,Y 185.992,Z 982.614,A -85,B 0,C 180,E1 9118.804,E2 9118.804} C_VEL
LIN {X 0,Y 180.028,Z 987.885,A -85,B 0,C 180,E1 9112.534,E2 9112.534} C_VEL
LIN {X 0,Y 175.492,Z 992.015,A -85,B 0,C 180,E1 9105.194,E2 9105.194} C_VEL
LIN {X 0,Y 173.176,Z 994.315,A -85,B 0,C 180,E1 9098.299,E2 9098.299} C_VEL
LIN {X 0,Y 172.304,Z 995.165,A -85,B 0,C 180,E1 9091.33,E2 9091.33} C_VEL
LIN {X 0,Y 172.718,Z 994.731,A -85,B 0,C 180,E1 9084.019,E2 9084.019} C_VEL
LIN {X 0,Y 174.526,Z 993.031,A -85,B 0,C 180,E1 9077.089,E2 9077.089} C_VEL
LIN {X 0,Y 178.145,Z 989.641,A -85,B 0,C 180,E1 9069.979,E2 9069.979} C_VEL
LIN {X 0,Y 183.823,Z 984.578,A -85,B 0,C 180,E1 9063.163,E2 9063.163} C_VEL
LIN {X 0,Y 191.51,Z 977.705,A -85,B 0,C 180,E1 9056.756,E2 9056.756} C_VEL
LIN {X 0,Y 200.172,Z 969.738,A -85,B 0,C 180,E1 9051.363,E2 9051.363} C_VEL
LIN {X 0,Y 210.267,Z 959.806,A -85,B 0,C 180,E1 9046.409,E2 9046.409} C_VEL
LIN {X 0,Y 220.448,Z 949.032,A -85,B 0,C 180,E1 9042.328,E2 9042.328} C_VEL
LIN {X 0,Y 230.911,Z 937.084,A -85,B 0,C 180,E1 9038.793,E2 9038.793} C_VEL
LIN {X 0,Y 242.091,Z 922.93,A -85,B 0,C 180,E1 9035.547,E2 9035.547} C_VEL
LIN {X 0,Y 252.457,Z 908.22,A -85,B 0,C 180,E1 9032.898,E2 9032.898} C_VEL
LIN {X 0,Y 262.896,Z 891.591,A -85,B 0,C 180,E1 9030.521,E2 9030.521} C_VEL
LIN {X 0,Y 272.551,Z 874.013,A -85,B 0,C 180,E1 9028.524,E2 9028.524} C_VEL
LIN {X 0,Y 281.268,Z 855.267,A -85,B 0,C 180,E1 9026.838,E2 9026.838} C_VEL
LIN {X 0,Y 288.969,Z 835.595,A -85,B 0,C 180,E1 9025.433,E2 9025.433} C_VEL
LIN {X 0,Y 295.389,Z 815.586,A -85,B 0,C 180,E1 9024.302,E2 9024.302} C_VEL
LIN {X 0,Y 300.6,Z 794.664,A -85,B 0,C 180,E1 9023.389,E2 9023.389} C_VEL
LIN {X 0,Y 304.347,Z 773.508,A -85,B 0,C 180,E1 9022.699,E2 9022.699} C_VEL
LIN {X 0,Y 307.358,Z 746.167,A -85,B 0,C 180,E1 9022.085,E2 9022.085} C_VEL
LIN {X 0,Y 320.98,Z 601.475,A -85,B 0,C 180,E1 9019.423,E2 9019.423} C_VEL
LIN {X 0,Y 317.973,Z 594.881,A -85,B 0,C 180,E1 9016.346,E2 9016.346} C_VEL
LIN {X 0,Y 316.05,Z 590.837,A -85,B 0,C 180,E1 9013.776,E2 9013.776} C_VEL
LIN {X 0,Y 314.814,Z 588.149,A -85,B 0,C 180,E1 9011.543,E2 9011.543} C_VEL
LIN {X 0,Y 313.594,Z 584.923,A -85,B 0,C 180,E1 9007.434,E2 9007.434} C_VEL
LIN {X 0,Y 313.819,Z 585.073,A -85,B 0,C 180,E1 9002.374,E2 9002.374} C_VEL
LIN {X 0,Y 313.88,Z 585.125,A -85,B 0,C 180,E1 9002.152,E2 9002.152} C_VEL
LIN {X 0,Y 314.157,Z 586.448,A -85,B 0,C 180,E1 9000.97,E2 9000.97} C_VEL
LIN {X 0,Y 314.41,Z 590.249,A -85,B 0,C 180,E1 8999.498,E2 8999.498} C_VEL
LIN {X 0,Y 315.088,Z 597.435,A -85,B 0,C 180,E1 8997.158,E2 8997.158} C_VEL
LIN {X 0,Y 315.661,Z 599.285,A -85,B 0,C 180,E1 8996.194,E2 8996.194} C_VEL
LIN {X 0,Y 318.168,Z 604.593,A -85,B 0,C 180,E1 8993.142,E2 8993.142} C_VEL
LIN {X 0,Y 320.026,Z 608.773,A -85,B 0,C 180,E1 8991.305,E2 8991.305} C_VEL
LIN {X 0,Y 301.881,Z 782.839,A -85,B 0,C 180,E1 8987.905,E2 8987.905} C_VEL
LIN {X 0,Y 297.889,Z 805.492,A -85,B 0,C 180,E1 8987.342,E2 8987.342} C_VEL
LIN {X 0,Y 292.182,Z 828.52,A -85,B 0,C 180,E1 8986.635,E2 8986.635} C_VEL
LIN {X 0,Y 285.203,Z 850.362,A -85,B 0,C 180,E1 8985.779,E2 8985.779} C_VEL
LIN {X 0,Y 277.317,Z 870.512,A -85,B 0,C 180,E1 8984.72,E2 8984.72} C_VEL
LIN {X 0,Y 267.771,Z 891.52,A -85,B 0,C 180,E1 8983.291,E2 8983.291} C_VEL
LIN {X 0,Y 258.069,Z 910.152,A -85,B 0,C 180,E1 8981.665,E2 8981.665} C_VEL
LIN {X 0,Y 247.016,Z 928.938,A -85,B 0,C 180,E1 8979.563,E2 8979.563} C_VEL
LIN {X 0,Y 235.284,Z 947.004,A -85,B 0,C 180,E1 8976.987,E2 8976.987} C_VEL
LIN {X 0,Y 223.641,Z 963.413,A -85,B 0,C 180,E1 8973.98,E2 8973.98} C_VEL
LIN {X 0,Y 211.487,Z 979.319,A -85,B 0,C 180,E1 8970.238,E2 8970.238} C_VEL
LIN {X 0,Y 199.661,Z 994.147,A -85,B 0,C 180,E1 8965.719,E2 8965.719} C_VEL
LIN {X 0,Y 188.997,Z 1007.167,A -85,B 0,C 180,E1 8960.569,E2 8960.569} C_VEL
LIN {X 0,Y 179.489,Z 1018.919,A -85,B 0,C 180,E1 8954.519,E2 8954.519} C_VEL
LIN {X 0,Y 171.761,Z 1029.222,A -85,B 0,C 180,E1 8947.658,E2 8947.658} C_VEL
LIN {X 0,Y 166.358,Z 1037.629,A -85,B 0,C 180,E1 8940.323,E2 8940.323} C_VEL
LIN {X 0,Y 163.263,Z 1044.25,A -85,B 0,C 180,E1 8932.695,E2 8932.695} C_VEL
LIN {X 0,Y 162.291,Z 1048.768,A -85,B 0,C 180,E1 8925.729,E2 8925.729} C_VEL
LIN {X 0,Y 162.575,Z 1051.8,A -85,B 0,C 180,E1 8918.845,E2 8918.845} C_VEL
LIN {X 0,Y 163.187,Z 1053.073,A -85,B 0,C 180,E1 8913.513,E2 8913.513} C_VEL
LIN {X 0,Y 163.34,Z 1053.31,A -85,B 0,C 180,E1 8908.948,E2 8908.948} C_VEL
LIN {X 0,Y 162.911,Z 1052.597,A -85,B 0,C 180,E1 8904.011,E2 8904.011} C_VEL
LIN {X 0,Y 162.362,Z 1050.668,A -85,B 0,C 180,E1 8898.274,E2 8898.274} C_VEL
LIN {X 0,Y 162.475,Z 1047.251,A -85,B 0,C 180,E1 8891.708,E2 8891.708} C_VEL
LIN {X 0,Y 164.469,Z 1041.275,A -85,B 0,C 180,E1 8883.654,E2 8883.654} C_VEL
LIN {X 0,Y 168.66,Z 1033.8,A -85,B 0,C 180,E1 8876.092,E2 8876.092} C_VEL
LIN {X 0,Y 175.178,Z 1024.438,A -85,B 0,C 180,E1 8868.975,E2 8868.975} C_VEL
LIN {X 0,Y 184.043,Z 1013.14,A -85,B 0,C 180,E1 8862.349,E2 8862.349} C_VEL
LIN {X 0,Y 194.408,Z 1000.506,A -85,B 0,C 180,E1 8856.647,E2 8856.647} C_VEL
LIN {X 0,Y 205.86,Z 986.34,A -85,B 0,C 180,E1 8851.79,E2 8851.79} C_VEL
LIN {X 0,Y 217.924,Z 970.85,A -85,B 0,C 180,E1 8847.685,E2 8847.685} C_VEL
LIN {X 0,Y 229.891,Z 954.603,A -85,B 0,C 180,E1 8844.331,E2 8844.331} C_VEL
LIN {X 0,Y 241.822,Z 936.93,A -85,B 0,C 180,E1 8841.516,E2 8841.516} C_VEL
LIN {X 0,Y 253.085,Z 918.549,A -85,B 0,C 180,E1 8839.227,E2 8839.227} C_VEL
LIN {X 0,Y 263.926,Z 898.874,A -85,B 0,C 180,E1 8837.315,E2 8837.315} C_VEL
LIN {X 0,Y 273.345,Z 879.271,A -85,B 0,C 180,E1 8835.84,E2 8835.84} C_VEL
LIN {X 0,Y 282.085,Z 858.151,A -85,B 0,C 180,E1 8834.61,E2 8834.61} C_VEL
LIN {X 0,Y 289.611,Z 836.592,A -85,B 0,C 180,E1 8833.664,E2 8833.664} C_VEL
LIN {X 0,Y 295.721,Z 814.414,A -85,B 0,C 180,E1 8832.924,E2 8832.924} C_VEL
LIN {X 0,Y 300.332,Z 791.556,A -85,B 0,C 180,E1 8832.311,E2 8832.311} C_VEL
LIN {X 0,Y 303.647,Z 766.005,A -85,B 0,C 180,E1 8831.755,E2 8831.755} C_VEL
LIN {X 0,Y 319.837,Z 608.46,A -85,B 0,C 180,E1 8828.68,E2 8828.68} C_VEL
LIN {X 0,Y 316.88,Z 602.047,A -85,B 0,C 180,E1 8825.613,E2 8825.613} C_VEL
LIN {X 0,Y 315.044,Z 598.22,A -85,B 0,C 180,E1 8823.183,E2 8823.183} C_VEL
LIN {X 0,Y 313.999,Z 596.196,A -85,B 0,C 180,E1 8821.459,E2 8821.459} C_VEL
LIN {X 0,Y 312.657,Z 592.916,A -85,B 0,C 180,E1 8817.8,E2 8817.8} C_VEL
LIN {X 0,Y 312.283,Z 592.648,A -85,B 0,C 180,E1 8813.006,E2 8813.006} C_VEL
LIN {X 0,Y 312.52,Z 593.252,A -85,B 0,C 180,E1 8811.536,E2 8811.536} C_VEL
LIN {X 0,Y 314.03,Z 596.983,A -85,B 0,C 180,E1 8807.495,E2 8807.495} C_VEL
LIN {X 0,Y 315.658,Z 600.655,A -85,B 0,C 180,E1 8804.945,E2 8804.945} C_VEL
LIN {X 0,Y 318.043,Z 605.909,A -85,B 0,C 180,E1 8802.15,E2 8802.15} C_VEL
LIN {X 0,Y 318.413,Z 607.009,A -85,B 0,C 180,E1 8801.745,E2 8801.745} C_VEL
LIN {X 0,Y 302.777,Z 766.662,A -85,B 0,C 180,E1 8798.827,E2 8798.827} C_VEL
LIN {X 0,Y 299.301,Z 788.269,A -85,B 0,C 180,E1 8798.202,E2 8798.202} C_VEL
LIN {X 0,Y 294.383,Z 809.64,A -85,B 0,C 180,E1 8797.368,E2 8797.368} C_VEL
LIN {X 0,Y 288.219,Z 830.139,A -85,B 0,C 180,E1 8796.326,E2 8796.326} C_VEL
LIN {X 0,Y 280.692,Z 849.953,A -85,B 0,C 180,E1 8795.035,E2 8795.035} C_VEL
LIN {X 0,Y 272.097,Z 868.87,A -85,B 0,C 180,E1 8793.481,E2 8793.481} C_VEL
LIN {X 0,Y 262.835,Z 886.38,A -85,B 0,C 180,E1 8791.682,E2 8791.682} C_VEL
LIN {X 0,Y 252.422,Z 903.347,A -85,B 0,C 180,E1 8789.49,E2 8789.49} C_VEL
LIN {X 0,Y 241.93,Z 918.371,A -85,B 0,C 180,E1 8787.032,E2 8787.032} C_VEL
LIN {X 0,Y 230.853,Z 932.622,A -85,B 0,C 180,E1 8784.089,E2 8784.089} C_VEL
LIN {X 0,Y 219.695,Z 945.493,A -85,B 0,C 180,E1 8780.687,E2 8780.687} C_VEL
LIN {X 0,Y 208.732,Z 956.964,A -85,B 0,C 180,E1 8776.728,E2 8776.728} C_VEL
LIN {X 0,Y 197.677,Z 967.629,A -85,B 0,C 180,E1 8771.887,E2 8771.887} C_VEL
LIN {X 0,Y 188.049,Z 976.361,A -85,B 0,C 180,E1 8766.549,E2 8766.549} C_VEL
LIN {X 0,Y 179.215,Z 983.877,A -85,B 0,C 180,E1 8760.141,E2 8760.141} C_VEL
LIN {X 0,Y 172.733,Z 989.258,A -85,B 0,C 180,E1 8753.541,E2 8753.541} C_VEL
LIN {X 0,Y 167.865,Z 993.385,A -85,B 0,C 180,E1 8745.902,E2 8745.902} C_VEL
LIN {X 0,Y 165.366,Z 995.682,A -85,B 0,C 180,E1 8738.694,E2 8738.694} C_VEL
LIN {X 0,Y 164.423,Z 996.53,A -85,B 0,C 180,E1 8731.394,E2 8731.394} C_VEL
LIN {X 0,Y 164.872,Z 996.097,A -85,B 0,C 180,E1 8723.733,E2 8723.733} C_VEL
LIN {X 0,Y 166.826,Z 994.401,A -85,B 0,C 180,E1 8716.482,E2 8716.482} C_VEL
LIN {X 0,Y 170.721,Z 991.012,A -85,B 0,C 180,E1 8709.068,E2 8709.068} C_VEL
LIN {X 0,Y 176.779,Z 985.954,A -85,B 0,C 180,E1 8702.001,E2 8702.001} C_VEL
LIN {X 0,Y 184.93,Z 979.085,A -85,B 0,C 180,E1 8695.409,E2 8695.409} C_VEL
LIN {X 0,Y 194.045,Z 971.128,A -85,B 0,C 180,E1 8689.902,E2 8689.902} C_VEL
LIN {X 0,Y 204.608,Z 961.197,A -85,B 0,C 180,E1 8684.881,E2 8684.881} C_VEL
LIN {X 0,Y 215.821,Z 949.792,A -85,B 0,C 180,E1 8680.554,E2 8680.554} C_VEL
LIN {X 0,Y 227.371,Z 936.938,A -85,B 0,C 180,E1 8676.837,E2 8676.837} C_VEL
LIN {X 0,Y 239.003,Z 922.606,A -85,B 0,C 180,E1 8673.642,E2 8673.642} C_VEL
LIN {X 0,Y 249.733,Z 907.616,A -85,B 0,C 180,E1 8671.041,E2 8671.041} C_VEL
LIN {X 0,Y 260.503,Z 890.625,A -85,B 0,C 180,E1 8668.713,E2 8668.713} C_VEL
LIN {X 0,Y 270.052,Z 873.397,A -85,B 0,C 180,E1 8666.836,E2 8666.836} C_VEL
LIN {X 0,Y 278.611,Z 855.322,A -85,B 0,C 180,E1 8665.262,E2 8665.262} C_VEL
LIN {X 0,Y 286.106,Z 836.503,A -85,B 0,C 180,E1 8663.954,E2 8663.954} C_VEL
LIN {X 0,Y 292.675,Z 816.517,A -85,B 0,C 180,E1 8662.846,E2 8662.846} C_VEL
LIN {X 0,Y 298.007,Z 795.635,A -85,B 0,C 180,E1 8661.952,E2 8661.952} C_VEL
LIN {X 0,Y 301.872,Z 774.447,A -85,B 0,C 180,E1 8661.271,E2 8661.271} C_VEL
LIN {X 0,Y 304.917,Z 747.841,A -85,B 0,C 180,E1 8660.678,E2 8660.678} C_VEL
LIN {X 0,Y 318.612,Z 606.962,A -85,B 0,C 180,E1 8658.148,E2 8658.148} C_VEL
LIN {X 0,Y 316.12,Z 601.402,A -85,B 0,C 180,E1 8655.305,E2 8655.305} C_VEL
LIN {X 0,Y 314.72,Z 598.256,A -85,B 0,C 180,E1 8653.224,E2 8653.224} C_VEL
LIN {X 0,Y 313.691,Z 595.896,A -85,B 0,C 180,E1 8651.212,E2 8651.212} C_VEL
LIN {X 0,Y 312.607,Z 592.854,A -85,B 0,C 180,E1 8647.351,E2 8647.351} C_VEL
LIN {X 0,Y 312.845,Z 593.017,A -85,B 0,C 180,E1 8642.382,E2 8642.382} C_VEL
LIN {X 0,Y 314.9,Z 597.66,A -85,B 0,C 180,E1 8637.362,E2 8637.362} C_VEL
LIN {X 0,Y 315.661,Z 599.285,A -85,B 0,C 180,E1 8636.194,E2 8636.194} C_VEL
LIN {X 0,Y 316.099,Z 601.146,A -85,B 0,C 180,E1 8635.465,E2 8635.465} C_VEL
LIN {X 0,Y 316.51,Z 606.801,A -85,B 0,C 180,E1 8634.356,E2 8634.356} C_VEL
LIN {X 0,Y 316.985,Z 612.011,A -85,B 0,C 180,E1 8633.343,E2 8633.343} C_VEL
LIN {X 0,Y 317.481,Z 613.77,A -85,B 0,C 180,E1 8632.746,E2 8632.746} C_VEL
LIN {X 0,Y 317.589,Z 614.326,A -85,B 0,C 180,E1 8632.602,E2 8632.602} C_VEL
LIN {X 0,Y 299.71,Z 782.174,A -85,B 0,C 180,E1 8629.385,E2 8629.385} C_VEL
LIN {X 0,Y 295.644,Z 804.832,A -85,B 0,C 180,E1 8628.837,E2 8628.837} C_VEL
LIN {X 0,Y 289.88,Z 827.703,A -85,B 0,C 180,E1 8628.159,E2 8628.159} C_VEL
LIN {X 0,Y 282.783,Z 849.549,A -85,B 0,C 180,E1 8627.338,E2 8627.338} C_VEL
LIN {X 0,Y 274.687,Z 869.813,A -85,B 0,C 180,E1 8626.315,E2 8626.315} C_VEL
LIN {X 0,Y 265.053,Z 890.543,A -85,B 0,C 180,E1 8624.954,E2 8624.954} C_VEL
LIN {X 0,Y 255.063,Z 909.266,A -85,B 0,C 180,E1 8623.372,E2 8623.372} C_VEL
LIN {X 0,Y 243.771,Z 927.922,A -85,B 0,C 180,E1 8621.342,E2 8621.342} C_VEL
LIN {X 0,Y 231.631,Z 946.043,A -85,B 0,C 180,E1 8618.811,E2 8618.811} C_VEL
LIN {X 0,Y 219.653,Z 962.327,A -85,B 0,C 180,E1 8615.878,E2 8615.878} C_VEL
LIN {X 0,Y 206.938,Z 978.286,A -85,B 0,C 180,E1 8612.154,E2 8612.154} C_VEL
LIN {X 0,Y 194.314,Z 993.335,A -85,B 0,C 180,E1 8607.553,E2 8607.553} C_VEL
LIN {X 0,Y 182.558,Z 1006.948,A -85,B 0,C 180,E1 8602.063,E2 8602.063} C_VEL
LIN {X 0,Y 172.629,Z 1018.415,A -85,B 0,C 180,E1 8595.907,E2 8595.907} C_VEL
LIN {X 0,Y 164.088,Z 1029.001,A -85,B 0,C 180,E1 8588.428,E2 8588.428} C_VEL
LIN {X 0,Y 158.45,Z 1037.264,A -85,B 0,C 180,E1 8580.739,E2 8580.739} C_VEL
LIN {X 0,Y 155.353,Z 1043.401,A -85,B 0,C 180,E1 8573.025,E2 8573.025} C_VEL
LIN {X 0,Y 154.338,Z 1047.97,A -85,B 0,C 180,E1 8565.403,E2 8565.403} C_VEL
LIN {X 0,Y 154.695,Z 1050.615,A -85,B 0,C 180,E1 8558.549,E2 8558.549} C_VEL
LIN {X 0,Y 155.313,Z 1051.74,A -85,B 0,C 180,E1 8553.322,E2 8553.322} C_VEL
LIN {X 0,Y 155.454,Z 1051.944,A -85,B 0,C 180,E1 8548.894,E2 8548.894} C_VEL
LIN {X 0,Y 155.014,Z 1051.31,A -85,B 0,C 180,E1 8544.076,E2 8544.076} C_VEL
LIN {X 0,Y 154.404,Z 1049.258,A -85,B 0,C 180,E1 8537.661,E2 8537.661} C_VEL
LIN {X 0,Y 154.648,Z 1045.804,A -85,B 0,C 180,E1 8530.722,E2 8530.722} C_VEL
LIN {X 0,Y 156.947,Z 1039.831,A -85,B 0,C 180,E1 8522.313,E2 8522.313} C_VEL
LIN {X 0,Y 161.634,Z 1032.357,A -85,B 0,C 180,E1 8514.445,E2 8514.445} C_VEL
LIN {X 0,Y 168.802,Z 1022.938,A -85,B 0,C 180,E1 8507.064,E2 8507.064} C_VEL
LIN {X 0,Y 178.342,Z 1011.644,A -85,B 0,C 180,E1 8500.317,E2 8500.317} C_VEL
LIN {X 0,Y 189.398,Z 998.966,A -85,B 0,C 180,E1 8494.558,E2 8494.558} C_VEL
LIN {X 0,Y 201.465,Z 984.794,A -85,B 0,C 180,E1 8489.712,E2 8489.712} C_VEL
LIN {X 0,Y 214.081,Z 969.273,A -85,B 0,C 180,E1 8485.656,E2 8485.656} C_VEL
LIN {X 0,Y 226.514,Z 952.979,A -85,B 0,C 180,E1 8482.367,E2 8482.367} C_VEL
LIN {X 0,Y 238.597,Z 935.653,A -85,B 0,C 180,E1 8479.677,E2 8479.677} C_VEL
LIN {X 0,Y 250.44,Z 916.826,A -85,B 0,C 180,E1 8477.408,E2 8477.408} C_VEL
LIN {X 0,Y 261.559,Z 897.032,A -85,B 0,C 180,E1 8475.565,E2 8475.565} C_VEL
LIN {X 0,Y 271.193,Z 877.357,A -85,B 0,C 180,E1 8474.149,E2 8474.149} C_VEL
LIN {X 0,Y 279.791,Z 856.837,A -85,B 0,C 180,E1 8473.01,E2 8473.01} C_VEL
LIN {X 0,Y 287.363,Z 835.439,A -85,B 0,C 180,E1 8472.115,E2 8472.115} C_VEL
LIN {X 0,Y 293.536,Z 813.333,A -85,B 0,C 180,E1 8471.408,E2 8471.408} C_VEL
LIN {X 0,Y 298.19,Z 790.494,A -85,B 0,C 180,E1 8470.816,E2 8470.816} C_VEL
LIN {X 0,Y 301.599,Z 764.436,A -85,B 0,C 180,E1 8470.264,E2 8470.264} C_VEL
LIN {X 0,Y 317.405,Z 613.857,A -85,B 0,C 180,E1 8467.375,E2 8467.375} C_VEL
LIN {X 0,Y 314.656,Z 607.626,A -85,B 0,C 180,E1 8464.099,E2 8464.099} C_VEL
LIN {X 0,Y 312.997,Z 604.217,A -85,B 0,C 180,E1 8461.464,E2 8461.464} C_VEL
LIN {X 0,Y 311.616,Z 600.815,A -85,B 0,C 180,E1 8457.609,E2 8457.609} C_VEL
LIN {X 0,Y 311.368,Z 600.634,A -85,B 0,C 180,E1 8452.62,E2 8452.62} C_VEL
LIN {X 0,Y 312.442,Z 603.683,A -85,B 0,C 180,E1 8448.743,E2 8448.743} C_VEL
LIN {X 0,Y 314.238,Z 607.907,A -85,B 0,C 180,E1 8445.535,E2 8445.535} C_VEL
LIN {X 0,Y 316.162,Z 612.385,A -85,B 0,C 180,E1 8443.073,E2 8443.073} C_VEL
LIN {X 0,Y 300.544,Z 767.433,A -85,B 0,C 180,E1 8440.279,E2 8440.279} C_VEL
LIN {X 0,Y 296.972,Z 789.068,A -85,B 0,C 180,E1 8439.665,E2 8439.665} C_VEL
LIN {X 0,Y 291.891,Z 810.598,A -85,B 0,C 180,E1 8438.842,E2 8438.842} C_VEL
LIN {X 0,Y 285.713,Z 830.699,A -85,B 0,C 180,E1 8437.845,E2 8437.845} C_VEL
LIN {X 0,Y 278.294,Z 849.903,A -85,B 0,C 180,E1 8436.631,E2 8436.631} C_VEL
LIN {X 0,Y 269.093,Z 869.8,A -85,B 0,C 180,E1 8435.044,E2 8435.044} C_VEL
LIN {X 0,Y 259.667,Z 887.219,A -85,B 0,C 180,E1 8433.295,E2 8433.295} C_VEL
LIN {X 0,Y 249.489,Z 903.423,A -85,B 0,C 180,E1 8431.254,E2 8431.254} C_VEL
LIN {X 0,Y 238.47,Z 918.899,A -85,B 0,C 180,E1 8428.797,E2 8428.797} C_VEL
LIN {X 0,Y 227.023,Z 933.266,A -85,B 0,C 180,E1 8425.894,E2 8425.894} C_VEL
LIN {X 0,Y 215.437,Z 946.201,A -85,B 0,C 180,E1 8422.526,E2 8422.526} C_VEL
LIN {X 0,Y 203.926,Z 957.849,A -85,B 0,C 180,E1 8418.553,E2 8418.553} C_VEL
LIN {X 0,Y 192.573,Z 968.394,A -85,B 0,C 180,E1 8413.804,E2 8413.804} C_VEL
LIN {X 0,Y 182.148,Z 977.413,A -85,B 0,C 180,E1 8408.281,E2 8408.281} C_VEL
LIN {X 0,Y 173.161,Z 984.625,A -85,B 0,C 180,E1 8402.088,E2 8402.088} C_VEL
LIN {X 0,Y 165.783,Z 990.411,A -85,B 0,C 180,E1 8394.972,E2 8394.972} C_VEL
LIN {X 0,Y 160.622,Z 994.486,A -85,B 0,C 180,E1 8387.386,E2 8387.386} C_VEL
LIN {X 0,Y 157.745,Z 996.878,A -85,B 0,C 180,E1 8379.854,E2 8379.854} C_VEL
LIN {X 0,Y 156.568,Z 997.858,A -85,B 0,C 180,E1 8372.196,E2 8372.196} C_VEL
LIN {X 0,Y 156.872,Z 997.635,A -85,B 0,C 180,E1 8364.514,E2 8364.514} C_VEL
LIN {X 0,Y 158.731,Z 996.065,A -85,B 0,C 180,E1 8356.893,E2 8356.893} C_VEL
LIN {X 0,Y 162.633,Z 992.917,A -85,B 0,C 180,E1 8349.109,E2 8349.109} C_VEL
LIN {X 0,Y 168.811,Z 988.131,A -85,B 0,C 180,E1 8341.716,E2 8341.716} C_VEL
LIN {X 0,Y 176.878,Z 981.802,A -85,B 0,C 180,E1 8335.052,E2 8335.052} C_VEL
LIN {X 0,Y 186.787,Z 973.555,A -85,B 0,C 180,E1 8329.006,E2 8329.006} C_VEL
LIN {X 0,Y 197.613,Z 963.94,A -85,B 0,C 180,E1 8323.883,E2 8323.883} C_VEL
LIN {X 0,Y 209.494,Z 952.509,A -85,B 0,C 180,E1 8319.359,E2 8319.359} C_VEL
LIN {X 0,Y 221.37,Z 939.966,A -85,B 0,C 180,E1 8315.609,E2 8315.609} C_VEL
LIN {X 0,Y 233.312,Z 925.807,A -85,B 0,C 180,E1 8312.391,E2 8312.391} C_VEL
LIN {X 0,Y 244.649,Z 910.708,A -85,B 0,C 180,E1 8309.718,E2 8309.718} C_VEL
LIN {X 0,Y 255.672,Z 894.128,A -85,B 0,C 180,E1 8307.41,E2 8307.41} C_VEL
LIN {X 0,Y 265.824,Z 876.591,A -85,B 0,C 180,E1 8305.481,E2 8305.481} C_VEL
LIN {X 0,Y 274.965,Z 857.972,A -85,B 0,C 180,E1 8303.86,E2 8303.86} C_VEL
LIN {X 0,Y 283.033,Z 838.506,A -85,B 0,C 180,E1 8302.512,E2 8302.512} C_VEL
LIN {X 0,Y 289.705,Z 819.043,A -85,B 0,C 180,E1 8301.44,E2 8301.44} C_VEL
LIN {X 0,Y 295.271,Z 797.977,A -85,B 0,C 180,E1 8300.543,E2 8300.543} C_VEL
LIN {X 0,Y 299.412,Z 776.505,A -85,B 0,C 180,E1 8299.852,E2 8299.852} C_VEL
LIN {X 0,Y 302.258,Z 753.769,A -85,B 0,C 180,E1 8299.328,E2 8299.328} C_VEL
LIN {X 0,Y 316.346,Z 612.511,A -85,B 0,C 180,E1 8296.811,E2 8296.811} C_VEL
LIN {X 0,Y 313.99,Z 606.875,A -85,B 0,C 180,E1 8293.63,E2 8293.63} C_VEL
LIN {X 0,Y 312.643,Z 603.79,A -85,B 0,C 180,E1 8291.063,E2 8291.063} C_VEL
LIN {X 0,Y 311.608,Z 600.777,A -85,B 0,C 180,E1 8287.189,E2 8287.189} C_VEL
LIN {X 0,Y 311.882,Z 600.999,A -85,B 0,C 180,E1 8282.297,E2 8282.297} C_VEL
LIN {X 0,Y 313.722,Z 605.45,A -85,B 0,C 180,E1 8277.626,E2 8277.626} C_VEL
LIN {X 0,Y 315.581,Z 609.567,A -85,B 0,C 180,E1 8274.911,E2 8274.911} C_VEL
LIN {X 0,Y 317.481,Z 613.77,A -85,B 0,C 180,E1 8272.746,E2 8272.746} C_VEL
LIN {X 0,Y 317.711,Z 615.497,A -85,B 0,C 180,E1 8272.388,E2 8272.388} C_VEL
LIN {X 0,Y 317.54,Z 619.026,A -85,B 0,C 180,E1 8272.167,E2 8272.167} C_VEL
LIN {X 0,Y 316.813,Z 624.241,A -85,B 0,C 180,E1 8272.203,E2 8272.203} C_VEL
LIN {X 0,Y 315.207,Z 632.139,A -85,B 0,C 180,E1 8272.659,E2 8272.659} C_VEL
LIN {X 0,Y 313.121,Z 642.237,A -85,B 0,C 180,E1 8273.302,E2 8273.302} C_VEL
LIN {X 0,Y 312.316,Z 647.493,A -85,B 0,C 180,E1 8273.407,E2 8273.407} C_VEL
LIN {X 0,Y 312.16,Z 648.819,A -85,B 0,C 180,E1 8273.393,E2 8273.393} C_VEL
LIN {X 0,Y 297.722,Z 781.659,A -85,B 0,C 180,E1 8270.883,E2 8270.883} C_VEL
LIN {X 0,Y 293.582,Z 804.266,A -85,B 0,C 180,E1 8270.352,E2 8270.352} C_VEL
LIN {X 0,Y 287.608,Z 827.479,A -85,B 0,C 180,E1 8269.688,E2 8269.688} C_VEL
LIN {X 0,Y 280.682,Z 848.433,A -85,B 0,C 180,E1 8268.934,E2 8268.934} C_VEL
LIN {X 0,Y 272.411,Z 868.798,A -85,B 0,C 180,E1 8267.956,E2 8267.956} C_VEL
LIN {X 0,Y 262.562,Z 889.57,A -85,B 0,C 180,E1 8266.649,E2 8266.649} C_VEL
LIN {X 0,Y 252.41,Z 908.164,A -85,B 0,C 180,E1 8265.139,E2 8265.139} C_VEL
LIN {X 0,Y 240.782,Z 926.887,A -85,B 0,C 180,E1 8263.17,E2 8263.17} C_VEL
LIN {X 0,Y 227.881,Z 945.53,A -85,B 0,C 180,E1 8260.622,E2 8260.622} C_VEL
LIN {X 0,Y 215.14,Z 962.247,A -85,B 0,C 180,E1 8257.647,E2 8257.647} C_VEL
LIN {X 0,Y 202.353,Z 977.589,A -85,B 0,C 180,E1 8254.066,E2 8254.066} C_VEL
LIN {X 0,Y 189.178,Z 992.519,A -85,B 0,C 180,E1 8249.486,E2 8249.486} C_VEL
LIN {X 0,Y 177.402,Z 1005.427,A -85,B 0,C 180,E1 8244.253,E2 8244.253} C_VEL
LIN {X 0,Y 166.767,Z 1016.911,A -85,B 0,C 180,E1 8238.026,E2 8238.026} C_VEL
LIN {X 0,Y 157.484,Z 1027.514,A -85,B 0,C 180,E1 8230.361,E2 8230.361} C_VEL
LIN {X 0,Y 151.238,Z 1035.794,A -85,B 0,C 180,E1 8222.378,E2 8222.378} C_VEL
LIN {X 0,Y 147.609,Z 1042.159,A -85,B 0,C 180,E1 8213.98,E2 8213.98} C_VEL
LIN {X 0,Y 146.41,Z 1046.885,A -85,B 0,C 180,E1 8205.447,E2 8205.447} C_VEL
LIN {X 0,Y 146.776,Z 1049.325,A -85,B 0,C 180,E1 8198.619,E2 8198.619} C_VEL
LIN {X 0,Y 147.44,Z 1050.408,A -85,B 0,C 180,E1 8193.11,E2 8193.11} C_VEL
LIN {X 0,Y 147.547,Z 1050.546,A -85,B 0,C 180,E1 8188.447,E2 8188.447} C_VEL
LIN {X 0,Y 147.002,Z 1049.792,A -85,B 0,C 180,E1 8183.226,E2 8183.226} C_VEL
LIN {X 0,Y 146.441,Z 1047.843,A -85,B 0,C 180,E1 8176.978,E2 8176.978} C_VEL
LIN {X 0,Y 146.835,Z 1044.38,A -85,B 0,C 180,E1 8169.679,E2 8169.679} C_VEL
LIN {X 0,Y 149.357,Z 1038.665,A -85,B 0,C 180,E1 8161.184,E2 8161.184} C_VEL
LIN {X 0,Y 154.171,Z 1031.636,A -85,B 0,C 180,E1 8153.369,E2 8153.369} C_VEL
LIN {X 0,Y 161.774,Z 1022.404,A -85,B 0,C 180,E1 8145.7,E2 8145.7} C_VEL
LIN {X 0,Y 171.827,Z 1011.315,A -85,B 0,C 180,E1 8138.762,E2 8138.762} C_VEL
LIN {X 0,Y 183.402,Z 998.796,A -85,B 0,C 180,E1 8132.905,E2 8132.905} C_VEL
LIN {X 0,Y 195.95,Z 984.813,A -85,B 0,C 180,E1 8128.023,E2 8128.023} C_VEL
LIN {X 0,Y 209.762,Z 968.624,A -85,B 0,C 180,E1 8123.766,E2 8123.766} C_VEL
LIN {X 0,Y 222.8,Z 952.2,A -85,B 0,C 180,E1 8120.489,E2 8120.489} C_VEL
LIN {X 0,Y 235.302,Z 934.838,A -85,B 0,C 180,E1 8117.854,E2 8117.854} C_VEL
LIN {X 0,Y 247.189,Z 916.522,A -85,B 0,C 180,E1 8115.699,E2 8115.699} C_VEL
LIN {X 0,Y 258.056,Z 897.857,A -85,B 0,C 180,E1 8113.989,E2 8113.989} C_VEL
LIN {X 0,Y 267.926,Z 878.259,A -85,B 0,C 180,E1 8112.608,E2 8112.608} C_VEL
LIN {X 0,Y 277.271,Z 856.669,A -85,B 0,C 180,E1 8111.439,E2 8111.439} C_VEL
LIN {X 0,Y 285.054,Z 835.194,A -85,B 0,C 180,E1 8110.574,E2 8110.574} C_VEL
LIN {X 0,Y 291.516,Z 812.427,A -85,B 0,C 180,E1 8109.874,E2 8109.874} C_VEL
LIN {X 0,Y 296.203,Z 789.756,A -85,B 0,C 180,E1 8109.307,E2 8109.307} C_VEL
LIN {X 0,Y 299.682,Z 763.648,A -85,B 0,C 180,E1 8108.769,E2 8108.769} C_VEL
LIN {X 0,Y 315.114,Z 619.543,A -85,B 0,C 180,E1 8106.056,E2 8106.056} C_VEL
LIN {X 0,Y 312.874,Z 614.296,A -85,B 0,C 180,E1 8103.022,E2 8103.022} C_VEL
LIN {X 0,Y 311.801,Z 611.926,A -85,B 0,C 180,E1 8101.102,E2 8101.102} C_VEL
LIN {X 0,Y 310.58,Z 608.714,A -85,B 0,C 180,E1 8097.416,E2 8097.416} C_VEL
LIN {X 0,Y 310.434,Z 608.609,A -85,B 0,C 180,E1 8092.411,E2 8092.411} C_VEL
LIN {X 0,Y 311.779,Z 612.53,A -85,B 0,C 180,E1 8088.062,E2 8088.062} C_VEL
LIN {X 0,Y 313.198,Z 616.105,A -85,B 0,C 180,E1 8085.581,E2 8085.581} C_VEL
LIN {X 0,Y 314.05,Z 618.271,A -85,B 0,C 180,E1 8084.401,E2 8084.401} C_VEL
LIN {X 0,Y 298.519,Z 768.101,A -85,B 0,C 180,E1 8081.754,E2 8081.754} C_VEL
LIN {X 0,Y 294.844,Z 789.825,A -85,B 0,C 180,E1 8081.151,E2 8081.151} C_VEL
LIN {X 0,Y 289.805,Z 810.833,A -85,B 0,C 180,E1 8080.371,E2 8080.371} C_VEL
LIN {X 0,Y 283.57,Z 830.766,A -85,B 0,C 180,E1 8079.415,E2 8079.415} C_VEL
LIN {X 0,Y 276.117,Z 849.852,A -85,B 0,C 180,E1 8078.254,E2 8078.254} C_VEL
LIN {X 0,Y 267.108,Z 869.168,A -85,B 0,C 180,E1 8076.778,E2 8076.778} C_VEL
LIN {X 0,Y 257.441,Z 886.844,A -85,B 0,C 180,E1 8075.078,E2 8075.078} C_VEL
LIN {X 0,Y 246.767,Z 903.542,A -85,B 0,C 180,E1 8073.051,E2 8073.051} C_VEL
LIN {X 0,Y 235.246,Z 919.418,A -85,B 0,C 180,E1 8070.612,E2 8070.612} C_VEL
LIN {X 0,Y 223.425,Z 933.908,A -85,B 0,C 180,E1 8067.759,E2 8067.759} C_VEL
LIN {X 0,Y 210.728,Z 947.629,A -85,B 0,C 180,E1 8064.229,E2 8064.229} C_VEL
LIN {X 0,Y 198.858,Z 959.183,A -85,B 0,C 180,E1 8060.29,E2 8060.29} C_VEL
LIN {X 0,Y 187.17,Z 969.59,A -85,B 0,C 180,E1 8055.588,E2 8055.588} C_VEL
LIN {X 0,Y 176.064,Z 978.741,A -85,B 0,C 180,E1 8049.921,E2 8049.921} C_VEL
LIN {X 0,Y 166.495,Z 986.003,A -85,B 0,C 180,E1 8043.538,E2 8043.538} C_VEL
LIN {X 0,Y 158.634,Z 991.784,A -85,B 0,C 180,E1 8036.181,E2 8036.181} C_VEL
LIN {X 0,Y 153.084,Z 995.858,A -85,B 0,C 180,E1 8028.271,E2 8028.271} C_VEL
LIN {X 0,Y 149.971,Z 998.246,A -85,B 0,C 180,E1 8020.37,E2 8020.37} C_VEL
LIN {X 0,Y 148.691,Z 999.224,A -85,B 0,C 180,E1 8012.312,E2 8012.312} C_VEL
LIN {X 0,Y 149.021,Z 999.001,A -85,B 0,C 180,E1 8004.224,E2 8004.224} C_VEL
LIN {X 0,Y 151.039,Z 997.433,A -85,B 0,C 180,E1 7996.213,E2 7996.213} C_VEL
LIN {X 0,Y 155.317,Z 994.244,A -85,B 0,C 180,E1 7987.976,E2 7987.976} C_VEL
LIN {X 0,Y 162.219,Z 989.239,A -85,B 0,C 180,E1 7980.049,E2 7980.049} C_VEL
LIN {X 0,Y 170.739,Z 982.942,A -85,B 0,C 180,E1 7973.321,E2 7973.321} C_VEL
LIN {X 0,Y 181.123,Z 974.743,A -85,B 0,C 180,E1 7967.234,E2 7967.234} C_VEL
LIN {X 0,Y 192.544,Z 965.037,A -85,B 0,C 180,E1 7962.048,E2 7962.048} C_VEL
LIN {X 0,Y 205.232,Z 953.263,A -85,B 0,C 180,E1 7957.428,E2 7957.428} C_VEL
LIN {X 0,Y 216.931,Z 941.337,A -85,B 0,C 180,E1 7953.898,E2 7953.898} C_VEL
LIN {X 0,Y 229.162,Z 927.296,A -85,B 0,C 180,E1 7950.735,E2 7950.735} C_VEL
LIN {X 0,Y 240.85,Z 912.217,A -85,B 0,C 180,E1 7948.094,E2 7948.094} C_VEL
LIN {X 0,Y 251.773,Z 896.342,A -85,B 0,C 180,E1 7945.903,E2 7945.903} C_VEL
LIN {X 0,Y 262.019,Z 879.155,A -85,B 0,C 180,E1 7944.029,E2 7944.029} C_VEL
LIN {X 0,Y 271.489,Z 860.622,A -85,B 0,C 180,E1 7942.421,E2 7942.421} C_VEL
LIN {X 0,Y 279.731,Z 841.603,A -85,B 0,C 180,E1 7941.106,E2 7941.106} C_VEL
LIN {X 0,Y 286.791,Z 821.734,A -85,B 0,C 180,E1 7940.018,E2 7940.018} C_VEL
LIN {X 0,Y 292.542,Z 801.031,A -85,B 0,C 180,E1 7939.136,E2 7939.136} C_VEL
LIN {X 0,Y 297.096,Z 778.837,A -85,B 0,C 180,E1 7938.418,E2 7938.418} C_VEL
LIN {X 0,Y 300.019,Z 757.169,A -85,B 0,C 180,E1 7937.911,E2 7937.911} C_VEL
LIN {X 0,Y 314.264,Z 618.279,A -85,B 0,C 180,E1 7935.501,E2 7935.501} C_VEL
LIN {X 0,Y 312.466,Z 613.909,A -85,B 0,C 180,E1 7932.756,E2 7932.756} C_VEL
LIN {X 0,Y 311.44,Z 611.383,A -85,B 0,C 180,E1 7930.545,E2 7930.545} C_VEL
LIN {X 0,Y 310.612,Z 608.701,A -85,B 0,C 180,E1 7927.027,E2 7927.027} C_VEL
LIN {X 0,Y 310.863,Z 608.949,A -85,B 0,C 180,E1 7922.397,E2 7922.397} C_VEL
LIN {X 0,Y 312.599,Z 613.369,A -85,B 0,C 180,E1 7917.801,E2 7917.801} C_VEL
LIN {X 0,Y 314.407,Z 617.538,A -85,B 0,C 180,E1 7915.075,E2 7915.075} C_VEL
LIN {X 0,Y 315.311,Z 619.959,A -85,B 0,C 180,E1 7913.918,E2 7913.918} C_VEL
LIN {X 0,Y 312.16,Z 648.819,A -85,B 0,C 180,E1 7913.393,E2 7913.393} C_VEL
LIN {X 0,Y 311.122,Z 656.512,A -85,B 0,C 180,E1 7913.432,E2 7913.432} C_VEL
LIN {X 0,Y 307.666,Z 677.07,A -85,B 0,C 180,E1 7914.194,E2 7914.194} C_VEL
LIN {X 0,Y 306.807,Z 683.673,A -85,B 0,C 180,E1 7914.212,E2 7914.212} C_VEL
LIN {X 0,Y 295.866,Z 781.749,A -85,B 0,C 180,E1 7912.388,E2 7912.388} C_VEL
LIN {X 0,Y 291.608,Z 804.248,A -85,B 0,C 180,E1 7911.875,E2 7911.875} C_VEL
LIN {X 0,Y 285.692,Z 826.777,A -85,B 0,C 180,E1 7911.255,E2 7911.255} C_VEL
LIN {X 0,Y 278.749,Z 847.473,A -85,B 0,C 180,E1 7910.546,E2 7910.546} C_VEL
LIN {X 0,Y 270.384,Z 867.736,A -85,B 0,C 180,E1 7909.626,E2 7909.626} C_VEL
LIN {X 0,Y 260.306,Z 888.596,A -85,B 0,C 180,E1 7908.375,E2 7908.375} C_VEL
LIN {X 0,Y 249.497,Z 907.949,A -85,B 0,C 180,E1 7906.863,E2 7906.863} C_VEL
LIN {X 0,Y 237.604,Z 926.515,A -85,B 0,C 180,E1 7904.964,E2 7904.964} C_VEL
LIN {X 0,Y 223.948,Z 945.568,A -85,B 0,C 180,E1 7902.405,E2 7902.405} C_VEL
LIN {X 0,Y 211.239,Z 961.654,A -85,B 0,C 180,E1 7899.587,E2 7899.587} C_VEL
LIN {X 0,Y 198.005,Z 976.889,A -85,B 0,C 180,E1 7896.064,E2 7896.064} C_VEL
LIN {X 0,Y 184.053,Z 991.936,A -85,B 0,C 180,E1 7891.443,E2 7891.443} C_VEL
LIN {X 0,Y 171.296,Z 1005.134,A -85,B 0,C 180,E1 7885.982,E2 7885.982} C_VEL
LIN {X 0,Y 160.12,Z 1016.479,A -85,B 0,C 180,E1 7879.626,E2 7879.626} C_VEL
LIN {X 0,Y 150.523,Z 1026.624,A -85,B 0,C 180,E1 7871.932,E2 7871.932} C_VEL
LIN {X 0,Y 143.626,Z 1034.994,A -85,B 0,C 180,E1 7863.346,E2 7863.346} C_VEL
LIN {X 0,Y 139.816,Z 1041.105,A -85,B 0,C 180,E1 7854.744,E2 7854.744} C_VEL
LIN {X 0,Y 138.491,Z 1045.627,A -85,B 0,C 180,E1 7845.923,E2 7845.923} C_VEL
LIN {X 0,Y 138.857,Z 1048.035,A -85,B 0,C 180,E1 7838.697,E2 7838.697} C_VEL
LIN {X 0,Y 139.529,Z 1049.036,A -85,B 0,C 180,E1 7833.286,E2 7833.286} C_VEL
LIN {X 0,Y 139.676,Z 1049.21,A -85,B 0,C 180,E1 7828.769,E2 7828.769} C_VEL
LIN {X 0,Y 139.111,Z 1048.538,A -85,B 0,C 180,E1 7823.396,E2 7823.396} C_VEL
LIN {X 0,Y 138.502,Z 1046.589,A -85,B 0,C 180,E1 7816.643,E2 7816.643} C_VEL
LIN {X 0,Y 138.989,Z 1043.156,A -85,B 0,C 180,E1 7808.919,E2 7808.919} C_VEL
LIN {X 0,Y 142.023,Z 1037.198,A -85,B 0,C 180,E1 7799.543,E2 7799.543} C_VEL
LIN {X 0,Y 147.761,Z 1029.781,A -85,B 0,C 180,E1 7791.001,E2 7791.001} C_VEL
LIN {X 0,Y 156.219,Z 1020.423,A -85,B 0,C 180,E1 7783.143,E2 7783.143} C_VEL
LIN {X 0,Y 167.727,Z 1008.61,A -85,B 0,C 180,E1 7775.832,E2 7775.832} C_VEL
LIN {X 0,Y 179.543,Z 996.607,A -85,B 0,C 180,E1 7770.324,E2 7770.324} C_VEL
LIN {X 0,Y 192.936,Z 982.329,A -85,B 0,C 180,E1 7765.475,E2 7765.475} C_VEL
LIN {X 0,Y 206.481,Z 967.038,A -85,B 0,C 180,E1 7761.593,E2 7761.593} C_VEL
LIN {X 0,Y 219.776,Z 950.838,A -85,B 0,C 180,E1 7758.456,E2 7758.456} C_VEL
LIN {X 0,Y 232.162,Z 934.153,A -85,B 0,C 180,E1 7755.999,E2 7755.999} C_VEL
LIN {X 0,Y 244.608,Z 915.513,A -85,B 0,C 180,E1 7753.877,E2 7753.877} C_VEL
LIN {X 0,Y 255.771,Z 896.762,A -85,B 0,C 180,E1 7752.23,E2 7752.23} C_VEL
LIN {X 0,Y 266.236,Z 876.348,A -85,B 0,C 180,E1 7750.862,E2 7750.862} C_VEL
LIN {X 0,Y 275.472,Z 855.232,A -85,B 0,C 180,E1 7749.785,E2 7749.785} C_VEL
LIN {X 0,Y 283.189,Z 834.201,A -85,B 0,C 180,E1 7748.986,E2 7748.986} C_VEL
LIN {X 0,Y 289.604,Z 811.927,A -85,B 0,C 180,E1 7748.331,E2 7748.331} C_VEL
LIN {X 0,Y 294.406,Z 789.139,A -85,B 0,C 180,E1 7747.782,E2 7747.782} C_VEL
LIN {X 0,Y 297.943,Z 763.129,A -85,B 0,C 180,E1 7747.26,E2 7747.26} C_VEL
LIN {X 0,Y 312.994,Z 625.266,A -85,B 0,C 180,E1 7744.718,E2 7744.718} C_VEL
LIN {X 0,Y 311.215,Z 620.95,A -85,B 0,C 180,E1 7741.933,E2 7741.933} C_VEL
LIN {X 0,Y 309.592,Z 616.657,A -85,B 0,C 180,E1 7737.408,E2 7737.408} C_VEL
LIN {X 0,Y 309.444,Z 616.528,A -85,B 0,C 180,E1 7732.573,E2 7732.573} C_VEL
LIN {X 0,Y 310.668,Z 620.365,A -85,B 0,C 180,E1 7728.301,E2 7728.301} C_VEL
LIN {X 0,Y 311.982,Z 623.828,A -85,B 0,C 180,E1 7725.902,E2 7725.902} C_VEL
LIN {X 0,Y 312.049,Z 624.381,A -85,B 0,C 180,E1 7725.746,E2 7725.746} C_VEL
LIN {X 0,Y 296.682,Z 768.872,A -85,B 0,C 180,E1 7723.245,E2 7723.245} C_VEL
LIN {X 0,Y 292.933,Z 790.506,A -85,B 0,C 180,E1 7722.66,E2 7722.66} C_VEL
LIN {X 0,Y 287.715,Z 811.789,A -85,B 0,C 180,E1 7721.891,E2 7721.891} C_VEL
LIN {X 0,Y 281.352,Z 831.697,A -85,B 0,C 180,E1 7720.963,E2 7720.963} C_VEL
LIN {X 0,Y 273.743,Z 850.773,A -85,B 0,C 180,E1 7719.836,E2 7719.836} C_VEL
LIN {X 0,Y 264.539,Z 870.098,A -85,B 0,C 180,E1 7718.403,E2 7718.403} C_VEL
LIN {X 0,Y 254.647,Z 887.787,A -85,B 0,C 180,E1 7716.751,E2 7716.751} C_VEL
LIN {X 0,Y 243.711,Z 904.511,A -85,B 0,C 180,E1 7714.775,E2 7714.775} C_VEL
LIN {X 0,Y 231.487,Z 920.899,A -85,B 0,C 180,E1 7712.308,E2 7712.308} C_VEL
LIN {X 0,Y 219.321,Z 935.345,A -85,B 0,C 180,E1 7709.501,E2 7709.501} C_VEL
LIN {X 0,Y 206.92,Z 948.328,A -85,B 0,C 180,E1 7706.215,E2 7706.215} C_VEL
LIN {X 0,Y 194.386,Z 960.149,A -85,B 0,C 180,E1 7702.258,E2 7702.258} C_VEL
LIN {X 0,Y 181.966,Z 970.784,A -85,B 0,C 180,E1 7697.478,E2 7697.478} C_VEL
LIN {X 0,Y 170.384,Z 979.875,A -85,B 0,C 180,E1 7691.816,E2 7691.816} C_VEL
LIN {X 0,Y 160.38,Z 987.067,A -85,B 0,C 180,E1 7685.436,E2 7685.436} C_VEL
LIN {X 0,Y 151.893,Z 992.934,A -85,B 0,C 180,E1 7677.864,E2 7677.864} C_VEL
LIN {X 0,Y 145.804,Z 997.093,A -85,B 0,C 180,E1 7669.635,E2 7669.635} C_VEL
LIN {X 0,Y 142.323,Z 999.518,A -85,B 0,C 180,E1 7661.345,E2 7661.345} C_VEL
LIN {X 0,Y 140.84,Z 1000.57,A -85,B 0,C 180,E1 7652.849,E2 7652.849} C_VEL
LIN {X 0,Y 141.071,Z 1000.475,A -85,B 0,C 180,E1 7644.713,E2 7644.713} C_VEL
LIN {X 0,Y 143.073,Z 998.991,A -85,B 0,C 180,E1 7636.255,E2 7636.255} C_VEL
LIN {X 0,Y 147.671,Z 995.84,A -85,B 0,C 180,E1 7627.298,E2 7627.298} C_VEL
LIN {X 0,Y 154.652,Z 991.152,A -85,B 0,C 180,E1 7619.286,E2 7619.286} C_VEL
LIN {X 0,Y 163.971,Z 984.667,A -85,B 0,C 180,E1 7611.984,E2 7611.984} C_VEL
LIN {X 0,Y 174.825,Z 976.541,A -85,B 0,C 180,E1 7605.753,E2 7605.753} C_VEL
LIN {X 0,Y 186.706,Z 966.959,A -85,B 0,C 180,E1 7600.496,E2 7600.496} C_VEL
LIN {X 0,Y 199.164,Z 955.982,A -85,B 0,C 180,E1 7596.073,E2 7596.073} C_VEL
LIN {X 0,Y 211.841,Z 943.558,A -85,B 0,C 180,E1 7592.343,E2 7592.343} C_VEL
LIN {X 0,Y 224.476,Z 929.629,A -85,B 0,C 180,E1 7589.188,E2 7589.188} C_VEL
LIN {X 0,Y 237.061,Z 913.98,A -85,B 0,C 180,E1 7586.458,E2 7586.458} C_VEL
LIN {X 0,Y 248.441,Z 897.938,A -85,B 0,C 180,E1 7584.278,E2 7584.278} C_VEL
LIN {X 0,Y 259.057,Z 880.571,A -85,B 0,C 180,E1 7582.424,E2 7582.424} C_VEL
LIN {X 0,Y 268.607,Z 862.402,A -85,B 0,C 180,E1 7580.881,E2 7580.881} C_VEL
LIN {X 0,Y 277.022,Z 843.605,A -85,B 0,C 180,E1 7579.604,E2 7579.604} C_VEL
LIN {X 0,Y 284.22,Z 823.899,A -85,B 0,C 180,E1 7578.544,E2 7578.544} C_VEL
LIN {X 0,Y 290.313,Z 802.816,A -85,B 0,C 180,E1 7577.658,E2 7577.658} C_VEL
LIN {X 0,Y 294.894,Z 781.636,A -85,B 0,C 180,E1 7576.976,E2 7576.976} C_VEL
LIN {X 0,Y 297.957,Z 760.292,A -85,B 0,C 180,E1 7576.472,E2 7576.472} C_VEL
LIN {X 0,Y 312.297,Z 624.217,A -85,B 0,C 180,E1 7574.139,E2 7574.139} C_VEL
LIN {X 0,Y 310.989,Z 620.791,A -85,B 0,C 180,E1 7571.781,E2 7571.781} C_VEL
LIN {X 0,Y 310.151,Z 618.679,A -85,B 0,C 180,E1 7569.651,E2 7569.651} C_VEL
LIN {X 0,Y 309.622,Z 616.625,A -85,B 0,C 180,E1 7566.863,E2 7566.863} C_VEL
LIN {X 0,Y 309.834,Z 616.82,A -85,B 0,C 180,E1 7562.59,E2 7562.59} C_VEL
LIN {X 0,Y 311.382,Z 621.03,A -85,B 0,C 180,E1 7558.16,E2 7558.16} C_VEL
LIN {X 0,Y 313.148,Z 625.351,A -85,B 0,C 180,E1 7555.33,E2 7555.33} C_VEL
LIN {X 0,Y 313.16,Z 625.878,A -85,B 0,C 180,E1 7555.248,E2 7555.248} C_VEL
LIN {X 0,Y 306.807,Z 683.673,A -85,B 0,C 180,E1 7554.212,E2 7554.212} C_VEL
LIN {X 0,Y 305.786,Z 691.367,A -85,B 0,C 180,E1 7554.256,E2 7554.256} C_VEL
LIN {X 0,Y 302.359,Z 711.921,A -85,B 0,C 180,E1 7555.04,E2 7555.04} C_VEL
LIN {X 0,Y 301.482,Z 718.523,A -85,B 0,C 180,E1 7555.065,E2 7555.065} C_VEL
LIN {X 0,Y 294.215,Z 781.807,A -85,B 0,C 180,E1 7553.911,E2 7553.911} C_VEL
LIN {X 0,Y 289.782,Z 804.512,A -85,B 0,C 180,E1 7553.41,E2 7553.41} C_VEL
LIN {X 0,Y 283.857,Z 826.504,A -85,B 0,C 180,E1 7552.829,E2 7552.829} C_VEL
LIN {X 0,Y 276.565,Z 847.768,A -85,B 0,C 180,E1 7552.134,E2 7552.134} C_VEL
LIN {X 0,Y 268.076,Z 867.826,A -85,B 0,C 180,E1 7551.262,E2 7551.262} C_VEL
LIN {X 0,Y 257.827,Z 888.479,A -85,B 0,C 180,E1 7550.072,E2 7550.072} C_VEL
LIN {X 0,Y 246.815,Z 907.719,A -85,B 0,C 180,E1 7548.626,E2 7548.626} C_VEL
LIN {X 0,Y 234.665,Z 926.141,A -85,B 0,C 180,E1 7546.805,E2 7546.805} C_VEL
LIN {X 0,Y 221.099,Z 944.512,A -85,B 0,C 180,E1 7544.417,E2 7544.417} C_VEL
LIN {X 0,Y 207.587,Z 961.026,A -85,B 0,C 180,E1 7541.599,E2 7541.599} C_VEL
LIN {X 0,Y 193.126,Z 977.038,A -85,B 0,C 180,E1 7537.931,E2 7537.931} C_VEL
LIN {X 0,Y 179.034,Z 991.473,A -85,B 0,C 180,E1 7533.464,E2 7533.464} C_VEL
LIN {X 0,Y 165.355,Z 1004.812,A -85,B 0,C 180,E1 7527.838,E2 7527.838} C_VEL
LIN {X 0,Y 153.514,Z 1016.139,A -85,B 0,C 180,E1 7521.3,E2 7521.3} C_VEL
LIN {X 0,Y 143.601,Z 1025.821,A -85,B 0,C 180,E1 7513.576,E2 7513.576} C_VEL
LIN {X 0,Y 136.079,Z 1034.159,A -85,B 0,C 180,E1 7504.456,E2 7504.456} C_VEL
LIN {X 0,Y 131.902,Z 1040.332,A -85,B 0,C 180,E1 7495.119,E2 7495.119} C_VEL
LIN {X 0,Y 130.563,Z 1044.534,A -85,B 0,C 180,E1 7486.003,E2 7486.003} C_VEL
LIN {X 0,Y 130.932,Z 1046.744,A -85,B 0,C 180,E1 7478.785,E2 7478.785} C_VEL
LIN {X 0,Y 131.659,Z 1047.704,A -85,B 0,C 180,E1 7473.047,E2 7473.047} C_VEL
LIN {X 0,Y 131.785,Z 1047.843,A -85,B 0,C 180,E1 7468.696,E2 7468.696} C_VEL
LIN {X 0,Y 131.2,Z 1047.249,A -85,B 0,C 180,E1 7463.436,E2 7463.436} C_VEL
LIN {X 0,Y 130.555,Z 1045.17,A -85,B 0,C 180,E1 7455.814,E2 7455.814} C_VEL
LIN {X 0,Y 131.244,Z 1041.712,A -85,B 0,C 180,E1 7447.609,E2 7447.609} C_VEL
LIN {X 0,Y 134.814,Z 1035.731,A -85,B 0,C 180,E1 7437.721,E2 7437.721} C_VEL
LIN {X 0,Y 141.234,Z 1028.3,A -85,B 0,C 180,E1 7428.822,E2 7428.822} C_VEL
LIN {X 0,Y 150.487,Z 1018.928,A -85,B 0,C 180,E1 7420.761,E2 7420.761} C_VEL
LIN {X 0,Y 162.236,Z 1007.682,A -85,B 0,C 180,E1 7413.687,E2 7413.687} C_VEL
LIN {X 0,Y 175.357,Z 995.072,A -85,B 0,C 180,E1 7407.896,E2 7407.896} C_VEL
LIN {X 0,Y 189.253,Z 980.947,A -85,B 0,C 180,E1 7403.179,E2 7403.179} C_VEL
LIN {X 0,Y 203.481,Z 965.483,A -85,B 0,C 180,E1 7399.36,E2 7399.36} C_VEL
LIN {X 0,Y 216.813,Z 949.772,A -85,B 0,C 180,E1 7396.418,E2 7396.418} C_VEL
LIN {X 0,Y 229.801,Z 932.756,A -85,B 0,C 180,E1 7394.005,E2 7394.005} C_VEL
LIN {X 0,Y 242.279,Z 914.506,A -85,B 0,C 180,E1 7392.019,E2 7392.019} C_VEL
LIN {X 0,Y 253.711,Z 895.711,A -85,B 0,C 180,E1 7390.444,E2 7390.444} C_VEL
LIN {X 0,Y 263.861,Z 876.318,A -85,B 0,C 180,E1 7389.202,E2 7389.202} C_VEL
LIN {X 0,Y 273.243,Z 855.436,A -85,B 0,C 180,E1 7388.179,E2 7388.179} C_VEL
LIN {X 0,Y 281.306,Z 833.965,A -85,B 0,C 180,E1 7387.4,E2 7387.4} C_VEL
LIN {X 0,Y 287.883,Z 811.496,A -85,B 0,C 180,E1 7386.771,E2 7386.771} C_VEL
LIN {X 0,Y 292.821,Z 788.511,A -85,B 0,C 180,E1 7386.239,E2 7386.239} C_VEL
LIN {X 0,Y 296.426,Z 762.503,A -85,B 0,C 180,E1 7385.733,E2 7385.733} C_VEL
LIN {X 0,Y 311.02,Z 631.224,A -85,B 0,C 180,E1 7383.367,E2 7383.367} C_VEL
LIN {X 0,Y 309.627,Z 627.658,A -85,B 0,C 180,E1 7380.74,E2 7380.74} C_VEL
LIN {X 0,Y 308.537,Z 624.52,A -85,B 0,C 180,E1 7377.027,E2 7377.027} C_VEL
LIN {X 0,Y 308.471,Z 624.518,A -85,B 0,C 180,E1 7372.55,E2 7372.55} C_VEL
LIN {X 0,Y 309.563,Z 628.197,A -85,B 0,C 180,E1 7368.542,E2 7368.542} C_VEL
LIN {X 0,Y 310.247,Z 630.264,A -85,B 0,C 180,E1 7367.111,E2 7367.111} C_VEL
LIN {X 0,Y 295.062,Z 769.535,A -85,B 0,C 180,E1 7364.757,E2 7364.757} C_VEL
LIN {X 0,Y 291.232,Z 791.161,A -85,B 0,C 180,E1 7364.188,E2 7364.188} C_VEL
LIN {X 0,Y 286.047,Z 812.019,A -85,B 0,C 180,E1 7363.462,E2 7363.462} C_VEL
LIN {X 0,Y 279.536,Z 832.067,A -85,B 0,C 180,E1 7362.563,E2 7362.563} C_VEL
LIN {X 0,Y 271.582,Z 851.693,A -85,B 0,C 180,E1 7361.446,E2 7361.446} C_VEL
LIN {X 0,Y 262.187,Z 871.028,A -85,B 0,C 180,E1 7360.059,E2 7360.059} C_VEL
LIN {X 0,Y 251.659,Z 889.422,A -85,B 0,C 180,E1 7358.389,E2 7358.389} C_VEL
LIN {X 0,Y 240.062,Z 906.646,A -85,B 0,C 180,E1 7356.393,E2 7356.393} C_VEL
LIN {X 0,Y 227.938,Z 922.38,A -85,B 0,C 180,E1 7354.06,E2 7354.06} C_VEL
LIN {X 0,Y 215.427,Z 936.782,A -85,B 0,C 180,E1 7351.308,E2 7351.308} C_VEL
LIN {X 0,Y 202.638,Z 949.757,A -85,B 0,C 180,E1 7348.07,E2 7348.07} C_VEL
LIN {X 0,Y 189.831,Z 961.392,A -85,B 0,C 180,E1 7344.208,E2 7344.208} C_VEL
LIN {X 0,Y 176.972,Z 971.972,A -85,B 0,C 180,E1 7339.478,E2 7339.478} C_VEL
LIN {X 0,Y 164.766,Z 981.106,A -85,B 0,C 180,E1 7333.767,E2 7333.767} C_VEL
LIN {X 0,Y 153.987,Z 988.445,A -85,B 0,C 180,E1 7327.147,E2 7327.147} C_VEL
LIN {X 0,Y 144.932,Z 994.31,A -85,B 0,C 180,E1 7319.329,E2 7319.329} C_VEL
LIN {X 0,Y 138.371,Z 998.463,A -85,B 0,C 180,E1 7310.737,E2 7310.737} C_VEL
LIN {X 0,Y 134.463,Z 1000.984,A -85,B 0,C 180,E1 7301.582,E2 7301.582} C_VEL
LIN {X 0,Y 132.937,Z 1001.954,A -85,B 0,C 180,E1 7292.587,E2 7292.587} C_VEL
LIN {X 0,Y 133.274,Z 1001.792,A -85,B 0,C 180,E1 7283.971,E2 7283.971} C_VEL
LIN {X 0,Y 135.564,Z 1000.264,A -85,B 0,C 180,E1 7275.04,E2 7275.04} C_VEL
LIN {X 0,Y 140.395,Z 997.21,A -85,B 0,C 180,E1 7266.05,E2 7266.05} C_VEL
LIN {X 0,Y 147.886,Z 992.527,A -85,B 0,C 180,E1 7257.716,E2 7257.716} C_VEL
LIN {X 0,Y 157.798,Z 986.04,A -85,B 0,C 180,E1 7250.21,E2 7250.21} C_VEL
LIN {X 0,Y 169.238,Z 977.925,A -85,B 0,C 180,E1 7243.881,E2 7243.881} C_VEL
LIN {X 0,Y 181.666,Z 968.352,A -85,B 0,C 180,E1 7238.597,E2 7238.597} C_VEL
LIN {X 0,Y 194.615,Z 957.393,A -85,B 0,C 180,E1 7234.192,E2 7234.192} C_VEL
LIN {X 0,Y 207.726,Z 944.976,A -85,B 0,C 180,E1 7230.504,E2 7230.504} C_VEL
LIN {X 0,Y 220.742,Z 931.082,A -85,B 0,C 180,E1 7227.403,E2 7227.403} C_VEL
LIN {X 0,Y 233.859,Z 915.235,A -85,B 0,C 180,E1 7224.695,E2 7224.695} C_VEL
LIN {X 0,Y 245.732,Z 898.887,A -85,B 0,C 180,E1 7222.535,E2 7222.535} C_VEL
LIN {X 0,Y 256.594,Z 881.501,A -85,B 0,C 180,E1 7220.738,E2 7220.738} C_VEL
LIN {X 0,Y 266.525,Z 862.955,A -85,B 0,C 180,E1 7219.217,E2 7219.217} C_VEL
LIN {X 0,Y 274.964,Z 844.439,A -85,B 0,C 180,E1 7218.005,E2 7218.005} C_VEL
LIN {X 0,Y 282.276,Z 824.818,A -85,B 0,C 180,E1 7216.984,E2 7216.984} C_VEL
LIN {X 0,Y 288.529,Z 803.629,A -85,B 0,C 180,E1 7216.122,E2 7216.122} C_VEL
LIN {X 0,Y 293.252,Z 782.223,A -85,B 0,C 180,E1 7215.454,E2 7215.454} C_VEL
LIN {X 0,Y 296.414,Z 760.631,A -85,B 0,C 180,E1 7214.959,E2 7214.959} C_VEL
LIN {X 0,Y 310.522,Z 630.205,A -85,B 0,C 180,E1 7212.79,E2 7212.79} C_VEL
LIN {X 0,Y 309.322,Z 627.023,A -85,B 0,C 180,E1 7210.053,E2 7210.053} C_VEL
LIN {X 0,Y 308.657,Z 624.57,A -85,B 0,C 180,E1 7206.884,E2 7206.884} C_VEL
LIN {X 0,Y 308.82,Z 624.712,A -85,B 0,C 180,E1 7202.784,E2 7202.784} C_VEL
LIN {X 0,Y 310.228,Z 628.821,A -85,B 0,C 180,E1 7198.431,E2 7198.431} C_VEL
LIN {X 0,Y 311.208,Z 631.543,A -85,B 0,C 180,E1 7196.602,E2 7196.602} C_VEL
LIN {X 0,Y 301.482,Z 718.523,A -85,B 0,C 180,E1 7195.065,E2 7195.065} C_VEL
LIN {X 0,Y 300.455,Z 726.214,A -85,B 0,C 180,E1 7195.116,E2 7195.116} C_VEL
LIN {X 0,Y 297.153,Z 746.763,A -85,B 0,C 180,E1 7195.934,E2 7195.934} C_VEL
LIN {X 0,Y 296.291,Z 753.366,A -85,B 0,C 180,E1 7195.967,E2 7195.967} C_VEL
LIN {X 0,Y 292.309,Z 784.308,A -85,B 0,C 180,E1 7195.4,E2 7195.4} C_VEL
LIN {X 0,Y 287.698,Z 806.885,A -85,B 0,C 180,E1 7194.916,E2 7194.916} C_VEL
LIN {X 0,Y 281.573,Z 828.334,A -85,B 0,C 180,E1 7194.365,E2 7194.365} C_VEL
LIN {X 0,Y 273.636,Z 850.314,A -85,B 0,C 180,E1 7193.662,E2 7193.662} C_VEL
LIN {X 0,Y 264.566,Z 871.046,A -85,B 0,C 180,E1 7192.775,E2 7192.775} C_VEL
LIN {X 0,Y 254.147,Z 890.961,A -85,B 0,C 180,E1 7191.631,E2 7191.631} C_VEL
LIN {X 0,Y 242.059,Z 910.974,A -85,B 0,C 180,E1 7190.119,E2 7190.119} C_VEL
LIN {X 0,Y 229.714,Z 928.984,A -85,B 0,C 180,E1 7188.335,E2 7188.335} C_VEL
LIN {X 0,Y 216.327,Z 946.184,A -85,B 0,C 180,E1 7186.078,E2 7186.078} C_VEL
LIN {X 0,Y 201.661,Z 963.166,A -85,B 0,C 180,E1 7183.122,E2 7183.122} C_VEL
LIN {X 0,Y 187.658,Z 977.994,A -85,B 0,C 180,E1 7179.677,E2 7179.677} C_VEL
LIN {X 0,Y 172.98,Z 992.225,A -85,B 0,C 180,E1 7175.162,E2 7175.162} C_VEL
LIN {X 0,Y 158.939,Z 1005.082,A -85,B 0,C 180,E1 7169.525,E2 7169.525} C_VEL
LIN {X 0,Y 146.129,Z 1016.538,A -85,B 0,C 180,E1 7162.534,E2 7162.534} C_VEL
LIN {X 0,Y 135.764,Z 1026.038,A -85,B 0,C 180,E1 7154.399,E2 7154.399} C_VEL
LIN {X 0,Y 128.151,Z 1033.82,A -85,B 0,C 180,E1 7144.995,E2 7144.995} C_VEL
LIN {X 0,Y 123.804,Z 1039.851,A -85,B 0,C 180,E1 7134.832,E2 7134.832} C_VEL
LIN {X 0,Y 122.626,Z 1043.604,A -85,B 0,C 180,E1 7125.609,E2 7125.609} C_VEL
LIN {X 0,Y 123.164,Z 1045.765,A -85,B 0,C 180,E1 7117.463,E2 7117.463} C_VEL
LIN {X 0,Y 123.861,Z 1046.446,A -85,B 0,C 180,E1 7111.85,E2 7111.85} C_VEL
LIN {X 0,Y 123.79,Z 1046.369,A -85,B 0,C 180,E1 7107.222,E2 7107.222} C_VEL
LIN {X 0,Y 123.007,Z 1045.441,A -85,B 0,C 180,E1 7101.115,E2 7101.115} C_VEL
LIN {X 0,Y 122.648,Z 1043.255,A -85,B 0,C 180,E1 7093.421,E2 7093.421} C_VEL
LIN {X 0,Y 124.376,Z 1038.847,A -85,B 0,C 180,E1 7083.244,E2 7083.244} C_VEL
